# B&R Automation Studio project Inzynierka_Kucharczyk_2018
Automation Studio 4.3.7.46 SP; technology packages: Acp10Arnc0 3.18.2, mapp 1.62.1

## Configuration Config1

CPU 4PP065.0571-P74F, AutomationRuntime G4.34, Build 4.1.2

### Task classes (Cpu.sw)
```
Cyclic#4:
  AxisCtrl <- Source.Code.AxisControl.AxisCtrl.prg
  Program <- Source.Code.Package1.Program.prg
NcDataObjects: acp10etxen <- acp10etxen.dob, gAxis01a <- gAxis01obj.gAxis01a.dob, gAxis01i <- gAxis01obj.gAxis01i.dob
VcDataObjects: Visu <- Source.Visu.Visu.dob
Libraries: MpAxis, MpCom, MpBase, NcGlobal, Acp10_MC, brsystem, Acp10man, sys_lib, Acp10par, runtime
```

### Hardware
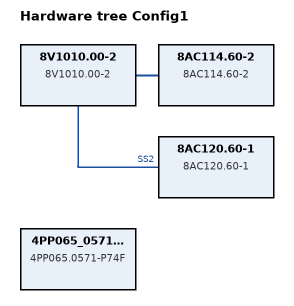
```
4PP065_0571_P74F : 4PP065.0571-P74F v1.0.3.0
  Connector IF5:
    ActivateDevice = 1
  ConfigurationID = Inzynierka_Kucharczyk_2018_Config1
  SimulationInaPort = 5900
  TimerDeviceType = EPLX2X
  TimerDevice = 4PP065_0571_P74F.IF4
  TaskClassIdleTime = 2000
  ActivateOpcUa = 1
  OpcUa_Security_AdminRole = Everyone
  OpcUaInformationModels_PV_Version = 1
  VcObjectName = Visu
  KeyMappingFile = VC\4PP065_0571_P74F.dis
8AC114.60-2 : 8AC114.60-2 v1.0.0.8  [SS -> 8V1010.00-2.SS1; PLK1 -> 4PP065_0571_P74F.IF4 [Cable Type=PowerlinkCable, Length=10, Version=1.0.0.1]]
8AC120.60-1 : 8AC120.60-1 v1.0.0.2  [SS -> 8V1010.00-2.SS2]
8V1010.00-2 : 8V1010.00-2 v1.0.0.2
  PoweredBy = DC
  BothEndSwitchesAreNormallyOpen_r1 = on
  QuickStopIsNormallyOpen_r1 = on
```

### Acp10cfg.ncc - 4PP065_0571_P74F/Motion/Acp10cfg.ncc
```
NcConfiguration (Version=3.18.2, NcSwId=Acp10)
  ACP10CF1_typ:
    cnt_nettrc_rec_drive = 150
    bufsize_trace_upload = 1200
    tc_nc_man_task = Cyclic #1
    glob_pv_as_ncobject = Yes
    ncsys_dl_broadcast = Yes
    ncsys_dl_acp_reset = Yes
    safemc_log_err_to_ax = Yes
    network_init:
      ncsw_init_execute = Yes
      automatic_execute = No
      node_nr_warning = Yes
      net_err_before_ncact = Yes
    nettrc:
      enter_parsecrec = Yes
      enter_ncaction = Yes
      save_ring_startidx = No
    cam_prof_download:
      cam_dat_dl_parallel = No
      tc_cam_dl_parallel = Task class for NC Manager task
    plk_if[0]:
      if_name = IF4
      tc_CycDat_PLCopen = Task class for NC Manager task
      mc_broadcast_extdat = No
```

### Acp10map.ncm - 4PP065_0571_P74F/Motion/Acp10map.ncm
```
NcMapping (NcSwId=Acp10)
  NcObject gAxis01 (ModuleId=8V1010.00-2, Type=ncAXIS, Channel=1, AcoposSimulation=Off, InitParameter=gAxis01i, AcoposParameter=gAxis01a, Disabled=FALSE, ModuleDisabled=FALSE)
  NcObject 8V1010.00-2_ncV_AXIS1 (ModuleId=8V1010.00-2, Type=ncV_AXIS, Channel=1, Disabled=TRUE, ModuleDisabled=FALSE)
```

### Config.mpaxisbasic - 4PP065_0571_P74F/mapp/Config.mpaxisbasic
```
Element gAxisBasic (Type=mpaxisbasic)
  AxisConfiguration = AxisWithConfiguration
    Axis:
      BaseType = 4
      MeasurementUnit = 1
    Drive:
      Controller:
        LoopFilters:
          [0]
          [1]
          [2]
```

## Logical view

Binary libraries used (declarations not repeated): operator, runtime, astime, AsIecCon, MpAxis 1.62.1, MpCom 1.62.1, MpBase 5.00.0, NcGlobal, Acp10_MC, brsystem, Acp10man, sys_lib, Acp10par, Acp10sim 3.18.2, ArEventLog, asstring, FileIO, ArProject

### Global.typ - Global data types
```iecst
TYPE
	Data_OPC_struct : 	STRUCT
		Zmienna1 : USINT;
		Zmienna2 : BOOL;
	END_STRUCT;
END_TYPE
```

### Global.var - Global variables
```iecst
VAR
	Zm_wyj : Data_OPC_struct;
	gAxis01 : ACP10AXIS_typ;
END_VAR
```


### Program Logical/Source/Code/AxisControl/AxisCtrl (IEC)

#### Main.st - Init, cyclic, exit code
```iecst
PROGRAM _INIT
	(* Task to initilization of drives *)
	Initialization;

END_PROGRAM

PROGRAM _CYCLIC

	AxesControl;

	Output_commands;
END_PROGRAM

PROGRAM _EXIT
	ExitAction;

END_PROGRAM
```

#### Initalization.st
```iecst
ACTION Initialization:

	_AxisCtrl.Internal.FunctionsBlock.MpAxisBasic_0.Enable := TRUE;
	_AxisCtrl.Internal.FunctionsBlock.MpAxisBasic_0.Axis   := ADR(gAxis01);
	_AxisCtrl.Internal.FunctionsBlock.MpAxisBasic_0.MpLink := ADR(gAxisBasic);
	_AxisCtrl.Internal.FunctionsBlock.MpAxisBasic_0.Parameters  := ADR(_AxisCtrl.Internal.Functions.MpAxisBasicParType_0);

END_ACTION
```

#### InputCmds.st
```iecst
ACTION Input_commands:

	(* ALL AXIS *)
	IF _AxisCtrl.Input.Commands.AllAxis.PowerOn THEN
		_AxisCtrl.Input.Commands.AllAxis.PowerOn := FALSE;
		_AxisCtrl.Output.Status.AxisStateMachine := POWER_ON;

	ELSIF _AxisCtrl.Input.Commands.AllAxis.PowerOff THEN
		_AxisCtrl.Input.Commands.AllAxis.PowerOff := FALSE;
		_AxisCtrl.Output.Status.AxisStateMachine := POWER_OFF;

	ELSIF _AxisCtrl.Input.Commands.AllAxis.Home THEN
		_AxisCtrl.Input.Commands.AllAxis.Home := FALSE;
		_AxisCtrl.Output.Status.AxisStateMachine := HOME;

	ELSIF _AxisCtrl.Input.Commands.AllAxis.StopOn THEN
		_AxisCtrl.Input.Commands.AllAxis.StopOn := FALSE;
		_AxisCtrl.Output.Status.AxisStateMachine := STOP_ON;

	ELSIF _AxisCtrl.Input.Commands.AllAxis.StopOff THEN
		_AxisCtrl.Input.Commands.AllAxis.StopOff := FALSE;
		_AxisCtrl.Output.Status.AxisStateMachine := STOP_OFF;

	ELSIF _AxisCtrl.Input.Commands.AllAxis.MoveAbsolute THEN
		_AxisCtrl.Input.Commands.AllAxis.MoveAbsolute := FALSE;
		_AxisCtrl.Output.Status.AxisStateMachine := MOVE_ABSOLUTE;

	ELSIF _AxisCtrl.Input.Commands.AllAxis.MoveVelocity THEN
		_AxisCtrl.Input.Commands.AllAxis.MoveVelocity := FALSE;
		_AxisCtrl.Output.Status.AxisStateMachine := MOVE_VELOCITY;

	ELSIF _AxisCtrl.Input.Commands.AllAxis.MoveAdditive THEN
		_AxisCtrl.Input.Commands.AllAxis.MoveAdditive := FALSE;
		_AxisCtrl.Output.Status.AxisStateMachine := MOVE_ADDITIVE;

	ELSIF _AxisCtrl.Input.Commands.AllAxis.JogPositive THEN
		_AxisCtrl.Output.Status.AxisStateMachine := JOG;

	ELSIF _AxisCtrl.Input.Commands.AllAxis.JogNegative THEN
		_AxisCtrl.Output.Status.AxisStateMachine := JOG;

	ELSIF _AxisCtrl.Input.Commands.AllAxis.ErrorReset THEN
		_AxisCtrl.Input.Commands.AllAxis.ErrorReset := FALSE;
		_AxisCtrl.Output.Status.AxisStateMachine := ERROR_RESET;

	(* SINGLE AXIS *)
	ELSIF _AxisCtrl.Input.Commands.SingleAxis.PowerOn THEN
		_AxisCtrl.Input.Commands.SingleAxis.PowerOn := FALSE;
		_AxisCtrl.Output.Status.AxisStateMachine := POWER_ON;

	ELSIF _AxisCtrl.Input.Commands.SingleAxis.PowerOff THEN
		_AxisCtrl.Input.Commands.SingleAxis.PowerOff := FALSE;
		_AxisCtrl.Output.Status.AxisStateMachine := POWER_OFF;

	ELSIF _AxisCtrl.Input.Commands.SingleAxis.Home THEN
		_AxisCtrl.Input.Commands.SingleAxis.Home := FALSE;
		_AxisCtrl.Output.Status.AxisStateMachine := HOME;

	ELSIF _AxisCtrl.Input.Commands.SingleAxis.StopOn THEN
		_AxisCtrl.Input.Commands.SingleAxis.StopOn := FALSE;
		_AxisCtrl.Output.Status.AxisStateMachine := STOP_ON;

	ELSIF _AxisCtrl.Input.Commands.SingleAxis.StopOff THEN
		_AxisCtrl.Input.Commands.SingleAxis.StopOff := FALSE;
		_AxisCtrl.Output.Status.AxisStateMachine := STOP_OFF;

	ELSIF _AxisCtrl.Input.Commands.SingleAxis.MoveAbsolute THEN
		_AxisCtrl.Input.Commands.SingleAxis.MoveAbsolute := FALSE;
		_AxisCtrl.Output.Status.AxisStateMachine := MOVE_ABSOLUTE;

	ELSIF _AxisCtrl.Input.Commands.SingleAxis.MoveVelocity THEN
		_AxisCtrl.Input.Commands.SingleAxis.MoveVelocity := FALSE;
		_AxisCtrl.Output.Status.AxisStateMachine := MOVE_VELOCITY;

	ELSIF _AxisCtrl.Input.Commands.SingleAxis.MoveAdditive THEN
		_AxisCtrl.Input.Commands.SingleAxis.MoveAdditive := FALSE;
		_AxisCtrl.Output.Status.AxisStateMachine := MOVE_ADDITIVE;

	ELSIF _AxisCtrl.Input.Commands.SingleAxis.JogPositive THEN
		_AxisCtrl.Output.Status.AxisStateMachine := JOG;

	ELSIF _AxisCtrl.Input.Commands.SingleAxis.JogNegative THEN
		_AxisCtrl.Output.Status.AxisStateMachine := JOG;

	ELSIF _AxisCtrl.Input.Commands.SingleAxis.ErrorReset THEN
		_AxisCtrl.Input.Commands.SingleAxis.ErrorReset := FALSE;
		_AxisCtrl.Output.Status.AxisStateMachine := ERROR_RESET;

	END_IF

END_ACTION
```

#### AxisControl.st
```iecst
ACTION AxesControl:

	CASE _AxisCtrl.Output.Status.AxisStateMachine OF
		WAIT_FOR_CMD:

			Input_commands;

		WAIT_FOR_ACTIVE:

		POWER_ON:

		POWER_OFF:

		HOME:

		STOP_ON:

		STOP_OFF:

		MOVE_ABSOLUTE:

		MOVE_VELOCITY:

		MOVE_ADDITIVE:

		JOG:

		ERROR_RESET:

	END_CASE;

END_ACTION
```

#### OutputCmds.st
```iecst
ACTION Output_commands:
	(* ALL AXES *)
	_AxisCtrl.Output.States.AllAxis.Active  := _AxisCtrl.Internal.FunctionsBlock.MpAxisBasic_0.Active;
	_AxisCtrl.Output.States.AllAxis.PowerOn := _AxisCtrl.Internal.FunctionsBlock.MpAxisBasic_0.PowerOn;
	_AxisCtrl.Output.States.AllAxis.IsHomed := _AxisCtrl.Internal.FunctionsBlock.MpAxisBasic_0.IsHomed;
	_AxisCtrl.Output.States.AllAxis.Stopped := _AxisCtrl.Internal.FunctionsBlock.MpAxisBasic_0.Stopped;
	_AxisCtrl.Output.States.AllAxis.InPosition := _AxisCtrl.Internal.FunctionsBlock.MpAxisBasic_0.InPosition;
	_AxisCtrl.Output.States.AllAxis.InVelocity := _AxisCtrl.Internal.FunctionsBlock.MpAxisBasic_0.InVelocity;
	_AxisCtrl.Output.States.AllAxis.MoveActive := _AxisCtrl.Internal.FunctionsBlock.MpAxisBasic_0.MoveActive;
	_AxisCtrl.Output.States.AllAxis.Error 	   := _AxisCtrl.Internal.FunctionsBlock.MpAxisBasic_0.Error;

	(* FIRST AXIS *)
	_AxisCtrl.Output.States.SingleAxis.Axis_0.Active  := _AxisCtrl.Internal.FunctionsBlock.MpAxisBasic_0.Active;
	_AxisCtrl.Output.States.SingleAxis.Axis_0.PowerOn := _AxisCtrl.Internal.FunctionsBlock.MpAxisBasic_0.PowerOn;
	_AxisCtrl.Output.States.SingleAxis.Axis_0.IsHomed := _AxisCtrl.Internal.FunctionsBlock.MpAxisBasic_0.IsHomed;
	_AxisCtrl.Output.States.SingleAxis.Axis_0.Stopped := _AxisCtrl.Internal.FunctionsBlock.MpAxisBasic_0.Stopped;
	_AxisCtrl.Output.States.SingleAxis.Axis_0.InPosition := _AxisCtrl.Internal.FunctionsBlock.MpAxisBasic_0.InPosition;
	_AxisCtrl.Output.States.SingleAxis.Axis_0.InVelocity := _AxisCtrl.Internal.FunctionsBlock.MpAxisBasic_0.InVelocity;
	_AxisCtrl.Output.States.SingleAxis.Axis_0.MoveActive := _AxisCtrl.Internal.FunctionsBlock.MpAxisBasic_0.MoveActive;
	_AxisCtrl.Output.States.SingleAxis.Axis_0.Error		 := _AxisCtrl.Internal.FunctionsBlock.MpAxisBasic_0.Error;
	_AxisCtrl.Output.States.SingleAxis.Axis_0.StatusID	 := _AxisCtrl.Internal.FunctionsBlock.MpAxisBasic_0.StatusID;

_AxisCtrl.Internal.FunctionsBlock.MpAxisBasic_0();
END_ACTION
```

#### Exit.st
```iecst
ACTION ExitAction:

END_ACTION
```

#### Axis1.st - not listed in the package file held
```iecst
ACTION Axis1:

	CASE _AxisCtrl.Output.Status.AxisStateMachine OF
		WAIT_FOR_CMD:

			IF _AxisCtrl.Input.Commands.SingleAxis.A1.PowerOn THEN
				_AxisCtrl.Input.Commands.SingleAxis.A1.PowerOn := FALSE;
				_AxisCtrl.Output.Status.AxisStateMachine := POWER_ON;

			ELSIF _AxisCtrl.Input.Commands.SingleAxis.A1.PowerOff THEN
				_AxisCtrl.Input.Commands.SingleAxis.A1.PowerOff := FALSE;
				_AxisCtrl.Output.Status.AxisStateMachine := POWER_OFF;

			ELSIF _AxisCtrl.Input.Commands.SingleAxis.A1.Home THEN
				_AxisCtrl.Input.Commands.SingleAxis.A1.Home := FALSE;
				_AxisCtrl.Output.Status.HomingStateMachine := PREPARE_HOME;
				_AxisCtrl.Output.Status.AxisStateMachine := HOME;

			ELSIF _AxisCtrl.Input.Commands.SingleAxis.A1.StopOn THEN
				_AxisCtrl.Input.Commands.SingleAxis.A1.StopOn := FALSE;
				_AxisCtrl.Output.Status.AxisStateMachine := STOP_ON;

			ELSIF _AxisCtrl.Input.Commands.SingleAxis.A1.StopOff THEN
				_AxisCtrl.Input.Commands.SingleAxis.A1.StopOff := FALSE;
				_AxisCtrl.Output.Status.AxisStateMachine := STOP_OFF;

			ELSIF _AxisCtrl.Input.Commands.SingleAxis.A1.MoveAbsolute THEN
				_AxisCtrl.Input.Commands.SingleAxis.A1.MoveAbsolute := FALSE;
				_AxisCtrl.Output.Status.AxisStateMachine := MOVE_ABSOLUTE;

			ELSIF _AxisCtrl.Input.Commands.SingleAxis.A1.MoveAbsoluteOff THEN
				_AxisCtrl.Input.Commands.SingleAxis.A1.MoveAbsoluteOff := FALSE;
				_AxisCtrl.Output.Status.AxisStateMachine := MOVE_ABSOLUTE_OFF;

			ELSIF _AxisCtrl.Input.Commands.SingleAxis.A1.MoveVelocity THEN
				_AxisCtrl.Input.Commands.SingleAxis.A1.MoveVelocity := FALSE;
				_AxisCtrl.Output.Status.AxisStateMachine := MOVE_VELOCITY;

			ELSIF _AxisCtrl.Input.Commands.SingleAxis.A1.MoveVelocityOff THEN
				_AxisCtrl.Input.Commands.SingleAxis.A1.MoveVelocityOff := FALSE;
				_AxisCtrl.Output.Status.AxisStateMachine := MOVE_VELOCITY_OFF;

			ELSIF _AxisCtrl.Input.Commands.SingleAxis.A1.MoveAdditive THEN
				_AxisCtrl.Input.Commands.SingleAxis.A1.MoveAdditive := FALSE;
				_AxisCtrl.Output.Status.AxisStateMachine := MOVE_ADDITIVE;

			ELSIF _AxisCtrl.Input.Commands.SingleAxis.A1.MoveAdditiveOff THEN
				_AxisCtrl.Input.Commands.SingleAxis.A1.MoveAdditiveOff := FALSE;
				_AxisCtrl.Output.Status.AxisStateMachine := MOVE_ADDITIVE_OFF;

			ELSIF _AxisCtrl.Input.Commands.SingleAxis.A1.JogPositive THEN
				_AxisCtrl.Output.Status.AxisStateMachine := JOG_POSITIVE;

			ELSIF _AxisCtrl.Input.Commands.SingleAxis.A1.JogNegative THEN
				_AxisCtrl.Output.Status.AxisStateMachine := JOG_NEGATIVE;

			ELSIF _AxisCtrl.Input.Commands.SingleAxis.A1.Update THEN
				_AxisCtrl.Input.Commands.SingleAxis.A1.Update := FALSE;
				_AxisCtrl.Internal.Functions.MpAxisBasicParType_0.Acceleration := _AxisCtrl.Input.Parameters.Acceleration;
				_AxisCtrl.Internal.Functions.MpAxisBasicParType_0.Deceleration := _AxisCtrl.Input.Parameters.Deceleration;
				_AxisCtrl.Internal.Functions.MpAxisBasicParType_0.Distance	   := _AxisCtrl.Input.Parameters.Distance;
				_AxisCtrl.Internal.Functions.MpAxisBasicParType_0.Position 	   := _AxisCtrl.Input.Parameters.Position;
				_AxisCtrl.Internal.Functions.MpAxisBasicParType_0.Velocity 	   := _AxisCtrl.Input.Parameters.Velocity;
			//	_AxisCtrl.Internal.Functions.MpAxisBasicParType_0.Torque.Limit  := _AxisCtrl.Input.Parameters.TorqueLimit;
			//	_AxisCtrl.Internal.Functions.MpAxisBasicParType_0.Torque.Window := _AxisCtrl.Input.Parameters.TorqueWindow;

				_AxisCtrl.Output.Status.AxisStateMachine := UPDATE_MP_AXIS_BASIC;

			ELSIF _AxisCtrl.Input.Commands.SingleAxis.A1.UpdateJogParams THEN
				_AxisCtrl.Input.Commands.SingleAxis.A1.UpdateJogParams := FALSE;
				_AxisCtrl.Internal.Functions.MpAxisBasicParType_0.Jog.Acceleration := _AxisCtrl.Input.Parameters.JogParams.Acceleration;
				_AxisCtrl.Internal.Functions.MpAxisBasicParType_0.Jog.Deceleration := _AxisCtrl.Input.Parameters.JogParams.Deceleration;
				_AxisCtrl.Internal.Functions.MpAxisBasicParType_0.Jog.LowerLimit   := _AxisCtrl.Input.Parameters.JogParams.LowerLimit;
			//	_AxisCtrl.Internal.Functions.MpAxisBasicParType_0.Jog.UpperLimit   := _AxisCtrl.Input.Parameters.JogParams.UpperLimit;
				_AxisCtrl.Internal.Functions.MpAxisBasicParType_0.Jog.Velocity     := _AxisCtrl.Input.Parameters.JogParams.JogVelocity;

				_AxisCtrl.Output.Status.AxisStateMachine := UPDATE_JOG_PARAMS;

				(* CYCLIC SET FUBS *)
			ELSIF _AxisCtrl.Input.Commands.SingleAxis.A1.TorqControl.CyclicPositionOn THEN
				_AxisCtrl.Input.Commands.SingleAxis.A1.TorqControl.CyclicPositionOn := FALSE;
				_AxisCtrl.Output.Status.AxisStateMachine := CYCLIC_POSITION_ON;

			ELSIF _AxisCtrl.Input.Commands.SingleAxis.A1.TorqControl.CyclicTorqueOn THEN
				_AxisCtrl.Input.Commands.SingleAxis.A1.TorqControl.CyclicTorqueOff := FALSE;
				_AxisCtrl.Output.Status.AxisStateMachine := CYCLIC_TORQUE_ON;

			ELSIF _AxisCtrl.Input.Commands.SingleAxis.A1.TorqControl.CyclicVelocityOn THEN
				_AxisCtrl.Input.Commands.SingleAxis.A1.TorqControl.CyclicVelocityOff := FALSE;
				_AxisCtrl.Output.Status.AxisStateMachine := CYCLIC_VELOCITY_ON;

			ELSIF _AxisCtrl.Input.Commands.SingleAxis.A1.TorqControl.CyclicPositionOff THEN
				_AxisCtrl.Input.Commands.SingleAxis.A1.TorqControl.CyclicPositionOff := FALSE;
				_AxisCtrl.Output.Status.AxisStateMachine := CYCLIC_POSITION_OFF;

			ELSIF _AxisCtrl.Input.Commands.SingleAxis.A1.TorqControl.CyclicTorqueOff THEN
				_AxisCtrl.Input.Commands.SingleAxis.A1.TorqControl.CyclicTorqueOff := FALSE;
				_AxisCtrl.Output.Status.AxisStateMachine := CYCLIC_TORQUE_OFF;

			ELSIF _AxisCtrl.Input.Commands.SingleAxis.A1.TorqControl.CyclicVelocityOff THEN
				_AxisCtrl.Input.Commands.SingleAxis.A1.TorqControl.CyclicVelocityOff := FALSE;
				_AxisCtrl.Output.Status.AxisStateMachine := CYCLIC_VELOCITY_OFF;

			ELSIF _AxisCtrl.Input.Commands.SingleAxis.A1.TorqControl.Update THEN

				_AxisCtrl.Internal.FunctionsBlock.TorqueControl.Position := _AxisCtrl.Input.Parameters.CyclicSetParameter.Position;
				_AxisCtrl.Internal.FunctionsBlock.TorqueControl.Torque 	 := _AxisCtrl.Input.Parameters.CyclicSetParameter.Torque;
				_AxisCtrl.Internal.FunctionsBlock.TorqueControl.Velocity := _AxisCtrl.Input.Parameters.CyclicSetParameter.Velocity;

				_AxisCtrl.Input.Commands.SingleAxis.A1.TorqControl.Update := FALSE;
				_AxisCtrl.Output.Status.AxisStateMachine := UPDATE_CYCLIC_SET;

			END_IF

		WAIT_FOR_ACTIVE:
			IF _AxisCtrl.Internal.FunctionsBlock.MpAxisBasic_0.Active THEN
				_AxisCtrl.Output.Status.AxisStateMachine := WAIT_FOR_CMD;
			ELSIF _AxisCtrl.Internal.FunctionsBlock.MpAxisBasic_0.Error THEN
				_AxisCtrl.Output.Status.AxisStateMachine := ERROR;
			END_IF

		POWER_ON:
			IF _AxisCtrl.Internal.FunctionsBlock.MpAxisBasic_0.PowerOn THEN
				_AxisCtrl.Output.Status.AxisStateMachine := WAIT_FOR_CMD;

			ELSIF _AxisCtrl.Internal.FunctionsBlock.MpAxisBasic_0.Error THEN
				_AxisCtrl.Internal.FunctionsBlock.MpAxisBasic_0.Power := FALSE;
				_AxisCtrl.Output.Status.AxisStateMachine := ERROR;

			ELSE
				_AxisCtrl.Internal.FunctionsBlock.MpAxisBasic_0.Power := TRUE;

			END_IF

		POWER_OFF:
			IF NOT _AxisCtrl.Internal.FunctionsBlock.MpAxisBasic_0.PowerOn THEN
				_AxisCtrl.Output.Status.AxisStateMachine := WAIT_FOR_CMD;

			ELSIF _AxisCtrl.Internal.FunctionsBlock.MpAxisBasic_0.Error THEN
				_AxisCtrl.Internal.FunctionsBlock.MpAxisBasic_0.Power := FALSE;
				_AxisCtrl.Output.Status.AxisStateMachine := ERROR;

			ELSE
				_AxisCtrl.Internal.FunctionsBlock.MpAxisBasic_0.Power := FALSE;
			END_IF

		HOME:
			CASE _AxisCtrl.Output.Status.HomingStateMachine OF
				PREPARE_HOME:
					_AxisCtrl.Internal.FunctionsBlock.MpAxisBasic_0.Home := FALSE;
					_AxisCtrl.Output.Status.HomingStateMachine := HOMING;
				HOMING:
					_AxisCtrl.Internal.FunctionsBlock.MpAxisBasic_0.Home := TRUE;
					IF _AxisCtrl.Internal.FunctionsBlock.MpAxisBasic_0.IsHomed THEN
						_AxisCtrl.Internal.FunctionsBlock.MpAxisBasic_0.Home := FALSE;
						_AxisCtrl.Output.Status.HomingStateMachine := EXIT_HOME;
					END_IF
				EXIT_HOME:
					_AxisCtrl.Output.Status.AxisStateMachine := WAIT_FOR_CMD;
					_AxisCtrl.Output.Status.HomingStateMachine := PREPARE_HOME;
			END_CASE;

		STOP_ON:
			IF _AxisCtrl.Internal.FunctionsBlock.MpAxisBasic_0.Stopped THEN
				_AxisCtrl.Output.Status.AxisStateMachine := WAIT_FOR_CMD;
			ELSIF _AxisCtrl.Internal.FunctionsBlock.MpAxisBasic_0.Error THEN
				_AxisCtrl.Internal.FunctionsBlock.MpAxisBasic_0.Stop := FALSE;
				_AxisCtrl.Output.Status.AxisStateMachine := ERROR;
			ELSE
				_AxisCtrl.Internal.FunctionsBlock.MpAxisBasic_0.Stop := TRUE;
			END_IF

		STOP_OFF:
			IF NOT _AxisCtrl.Internal.FunctionsBlock.MpAxisBasic_0.Stopped THEN
				_AxisCtrl.Output.Status.AxisStateMachine := WAIT_FOR_CMD;
			ELSIF _AxisCtrl.Internal.FunctionsBlock.MpAxisBasic_0.Error THEN
				_AxisCtrl.Internal.FunctionsBlock.MpAxisBasic_0.Stop := FALSE;
				_AxisCtrl.Output.Status.AxisStateMachine := ERROR;
			ELSE
				_AxisCtrl.Internal.FunctionsBlock.MpAxisBasic_0.Stop := FALSE;
			END_IF

		MOVE_ABSOLUTE:

			_AxisCtrl.Internal.FunctionsBlock.MpAxisBasic_0.MoveAbsolute := TRUE;
			_AxisCtrl.Output.Status.AxisStateMachine := WAIT_FOR_CMD;

		MOVE_ABSOLUTE_OFF:

			_AxisCtrl.Internal.FunctionsBlock.MpAxisBasic_0.MoveAbsolute := FALSE;
			_AxisCtrl.Output.Status.AxisStateMachine := WAIT_FOR_CMD;

		MOVE_VELOCITY:

			_AxisCtrl.Internal.FunctionsBlock.MpAxisBasic_0.MoveVelocity := TRUE;
			_AxisCtrl.Output.Status.AxisStateMachine := WAIT_FOR_CMD;

		MOVE_VELOCITY_OFF:

			_AxisCtrl.Internal.FunctionsBlock.MpAxisBasic_0.MoveVelocity := FALSE;
			_AxisCtrl.Output.Status.AxisStateMachine := WAIT_FOR_CMD;

		MOVE_ADDITIVE:

			_AxisCtrl.Internal.FunctionsBlock.MpAxisBasic_0.MoveAdditive := TRUE;
			_AxisCtrl.Output.Status.AxisStateMachine := WAIT_FOR_CMD;

		MOVE_ADDITIVE_OFF:

			_AxisCtrl.Internal.FunctionsBlock.MpAxisBasic_0.MoveAdditive := FALSE;
			_AxisCtrl.Output.Status.AxisStateMachine := WAIT_FOR_CMD;

		JOG_POSITIVE:
			IF NOT _AxisCtrl.Input.Commands.SingleAxis.A1.JogPositive THEN
				_AxisCtrl.Internal.FunctionsBlock.MpAxisBasic_0.JogPositive := FALSE;
				_AxisCtrl.Output.Status.AxisStateMachine := WAIT_FOR_CMD;
			ELSE
				_AxisCtrl.Internal.FunctionsBlock.MpAxisBasic_0.JogPositive := TRUE;
			END_IF

		JOG_NEGATIVE:
			IF NOT _AxisCtrl.Input.Commands.SingleAxis.A1.JogNegative THEN
				_AxisCtrl.Internal.FunctionsBlock.MpAxisBasic_0.JogNegative := FALSE;
				_AxisCtrl.Output.Status.AxisStateMachine := WAIT_FOR_CMD;
			ELSE
				_AxisCtrl.Internal.FunctionsBlock.MpAxisBasic_0.JogNegative := TRUE;
			END_IF

		UPDATE_MP_AXIS_BASIC:
			IF _AxisCtrl.Internal.FunctionsBlock.MpAxisBasic_0.UpdateDone THEN
				_AxisCtrl.Internal.FunctionsBlock.MpAxisBasic_0.Update := FALSE;
				_AxisCtrl.Output.Status.AxisStateMachine := WAIT_FOR_CMD;
			ELSE
				_AxisCtrl.Internal.FunctionsBlock.MpAxisBasic_0.Update := TRUE;
			END_IF

		UPDATE_JOG_PARAMS:
			IF _AxisCtrl.Internal.FunctionsBlock.MpAxisBasic_0.UpdateDone THEN
				_AxisCtrl.Internal.FunctionsBlock.MpAxisBasic_0.Update := FALSE;
				_AxisCtrl.Output.Status.AxisStateMachine := WAIT_FOR_CMD;
			ELSE
				_AxisCtrl.Internal.FunctionsBlock.MpAxisBasic_0.Update := TRUE;
			END_IF

		ERROR:
			IF _AxisCtrl.Input.Commands.SingleAxis.A1.ErrorReset OR _AxisCtrl.Input.Commands.SingleAxis.A1.TorqControl.ErrorReset THEN
				_AxisCtrl.Internal.FunctionsBlock.MpAxisBasic_0.ErrorReset := TRUE;
				_AxisCtrl.Internal.FunctionsBlock.TorqueControl.ErrorReset := TRUE;
				_AxisCtrl.Output.Status.AxisStateMachine := ERROR_RESET;
			END_IF

		ERROR_RESET:
			IF NOT _AxisCtrl.Output.States.SingleAxis.Axis_0.Error AND NOT _AxisCtrl.Internal.FunctionsBlock.TorqueControl.Error THEN
				_AxisCtrl.Internal.FunctionsBlock.MpAxisBasic_0.ErrorReset := FALSE;
				_AxisCtrl.Internal.FunctionsBlock.TorqueControl.ErrorReset := FALSE;
				_AxisCtrl.Output.Status.AxisStateMachine := WAIT_FOR_CMD;

			END_IF

		CYCLIC_POSITION_ON:

	    		_AxisCtrl.Internal.FunctionsBlock.TorqueControl.CyclicPosition := TRUE;
				_AxisCtrl.Output.Status.AxisStateMachine := WAIT_FOR_CMD;

		CYCLIC_POSITION_OFF:

				_AxisCtrl.Internal.FunctionsBlock.TorqueControl.CyclicPosition := FALSE;
				_AxisCtrl.Output.Status.AxisStateMachine := WAIT_FOR_CMD;

		CYCLIC_TORQUE_ON:

			_AxisCtrl.Internal.FunctionsBlock.TorqueControl.CyclicTorque := TRUE;
			_AxisCtrl.Output.Status.AxisStateMachine := WAIT_FOR_CMD;

		CYCLIC_TORQUE_OFF:

			_AxisCtrl.Internal.FunctionsBlock.TorqueControl.CyclicTorque := FALSE;
			_AxisCtrl.Output.Status.AxisStateMachine := WAIT_FOR_CMD;

		CYCLIC_VELOCITY_ON:

			_AxisCtrl.Internal.FunctionsBlock.TorqueControl.CyclicVelocity := TRUE;
			_AxisCtrl.Output.Status.AxisStateMachine := WAIT_FOR_CMD;

		CYCLIC_VELOCITY_OFF:

			_AxisCtrl.Internal.FunctionsBlock.TorqueControl.CyclicVelocity := FALSE;
			_AxisCtrl.Output.Status.AxisStateMachine := WAIT_FOR_CMD;

		UPDATE_CYCLIC_SET:
			IF _AxisCtrl.Internal.FunctionsBlock.TorqueControl.UpdateDone THEN
				_AxisCtrl.Internal.FunctionsBlock.TorqueControl.Update := FALSE;
				_AxisCtrl.Output.Status.AxisStateMachine := WAIT_FOR_CMD;
			ELSE
				_AxisCtrl.Internal.FunctionsBlock.TorqueControl.Update := TRUE;
			END_IF

	END_CASE;

END_ACTION
```

#### Axis2.st - not listed in the package file held
```iecst
ACTION Axis2:

END_ACTION
```

#### ErrorHandling.st - not listed in the package file held
```iecst
ACTION ErrorHandling:

	IF (_AxisCtrl.Internal.FunctionsBlock.MpAxisBasic_0.Error OR _AxisCtrl.Internal.FunctionsBlock.TorqueControl.Error) AND _AxisCtrl.Output.Status.AxisStateMachine <> ERROR_RESET THEN
		_AxisCtrl.Output.Status.AxisStateMachine := ERROR;
	END_IF

END_ACTION
```

#### Types.typ - Local data types
```iecst
(*Main structure*)

TYPE
	AxisCtrlType : 	STRUCT
		Input : AxisCtrlInpType; (*Inputs: ex. commands*)
		Internal : AxisCtrlInternalType; (*Fubs, funs*)
		Output : AxisCtrlOutType; (*States, status*)
	END_STRUCT;
END_TYPE

(**)
(*Inputs*)

TYPE
	AxisCtrlInpType : 	STRUCT
		Commands : {REDUND_UNREPLICABLE} AxisCtrlInpCmdType;
		Parameters : AxisCtrlInpParamsType;
	END_STRUCT;
END_TYPE

(**)

TYPE
	AxisCtrlInpCmdType : 	STRUCT
		SingleAxis : AxisCtrlInpCmdSigAxType;
		AllAxis : AxisCtrlInpCmdAllAxType;
	END_STRUCT;
	AxisCtrlInpParamsType : 	STRUCT
		Acceleration : REAL;
		Deceleration : REAL;
		Distance : REAL;
		Velocity : REAL;
		Position : REAL;
		JogParams : AxisCtrlInpParmsJogPType;
	END_STRUCT;
END_TYPE

(**)

TYPE
	AxisCtrlInpCmdSigAxType : 	STRUCT
		PowerOn : BOOL;
		PowerOff : BOOL;
		Home : BOOL;
		MoveVelocity : BOOL;
		MoveAdditive : BOOL;
		MoveAbsolute : BOOL;
		StopOn : BOOL;
		StopOff : BOOL;
		JogNegative : BOOL;
		JogPositive : BOOL;
		ErrorReset : BOOL;
	END_STRUCT;
	AxisCtrlInpCmdAllAxType : 	STRUCT
		PowerOn : BOOL;
		PowerOff : BOOL;
		Home : BOOL;
		MoveVelocity : BOOL;
		MoveAdditive : BOOL;
		MoveAbsolute : BOOL;
		StopOn : BOOL;
		StopOff : BOOL;
		JogNegative : BOOL;
		JogPositive : BOOL;
		ErrorReset : BOOL;
	END_STRUCT;
	AxisCtrlInpParmsJogPType : 	STRUCT
		JogVelocity : REAL;
		Acceleration : REAL;
		Deceleration : REAL;
		UpperLimit : LREAL;
		LowerLimit : LREAL;
	END_STRUCT;
END_TYPE

(**)
(*Internal*)

TYPE
	AxisCtrlInternalType : 	STRUCT
		FunctionsBlock : AxisCtrlInternalFubsType;
		Functions : AxisCtrlInternalFunsType;
	END_STRUCT;
END_TYPE

(**)

TYPE
	AxisCtrlInternalFubsType : 	STRUCT
		MpAxisBasic_0 : MpAxisBasic;
	END_STRUCT;
	AxisCtrlInternalFunsType : 	STRUCT
		MpAxisBasicParType_0 : MpAxisBasicParType;
	END_STRUCT;
END_TYPE

(**)
(*Output*)

TYPE
	AxisCtrlOutType : 	STRUCT
		Status : AxisCtrlOutStatusType;
		States : AxisCtrlOutStatesType;
	END_STRUCT;
	AxisCtrlOutStatusType : 	STRUCT
		HomingStateMachine : HomingEnum;
		AxisStateMachine : AxisCtrlEnum;
	END_STRUCT;
	AxisCtrlOutStatesType : 	STRUCT
		SingleAxis : AxisCtrlOutStatesSingType;
		AllAxis : AxisCtrlOutStatesAllType;
	END_STRUCT;
END_TYPE

(**)

TYPE
	AxisCtrlOutStatesAllType : 	STRUCT
		InPosition : BOOL;
		InVelocity : BOOL;
		UpdateDone : BOOL;
		Active : BOOL;
		Error : BOOL;
		Stopped : BOOL;
		MoveActive : BOOL;
		IsHomed : BOOL;
		PowerOn : BOOL;
	END_STRUCT;
	AxisCtrlOutStatesSingType : 	STRUCT
		Axis_0 : AxisCtrlOutStatesSingAxType;
		Axis_1 : AxisCtrlOutStatesSingAxType;
	END_STRUCT;
	AxisCtrlOutStatesSingAxType : 	STRUCT
		InPosition : BOOL;
		InVelocity : BOOL;
		StatusID : DINT;
		UpdateDone : BOOL;
		Active : BOOL;
		Error : BOOL;
		Stopped : BOOL;
		MoveActive : BOOL;
		IsHomed : BOOL;
		PowerOn : BOOL;
	END_STRUCT;
END_TYPE

(**)
(*Enumerators*)

TYPE
	HomingEnum :
		(
		PREPARE_HOME,
		HOMING,
		EXIT_HOME
		);
	AxisCtrlEnum :
		(
		WAIT_FOR_CMD,
		JOG,
		MOVE_ADDITIVE,
		MOVE_VELOCITY,
		MOVE_ABSOLUTE,
		STOP_OFF,
		STOP_ON,
		HOME,
		POWER_OFF,
		POWER_ON,
		WAIT_FOR_ACTIVE,
		ERROR_RESET
		);
END_TYPE
```

#### Variables.var - Local variables
```iecst
VAR
	_AxisCtrl : AxisCtrlType;
END_VAR
```

### Types.typ - not listed in the package file held
```iecst
(*Main structure*)

TYPE
	AxisCtrlType : 	STRUCT
		Input : AxisCtrlInpType; (*Inputs: ex. commands*)
		Internal : AxisCtrlInternalType; (*Fubs, funs*)
		Output : AxisCtrlOutType; (*States, status*)
	END_STRUCT;
END_TYPE

(**)
(*Inputs*)

TYPE
	AxisCtrlInpType : 	STRUCT
		Commands : {REDUND_UNREPLICABLE} AxisCtrlInpCmdType;
		Parameters : AxisCtrlInpParamsType;
	END_STRUCT;
END_TYPE

(**)

TYPE
	AxisCtrlInpCmdType : 	STRUCT
		SingleAxis : AxisCtrlInpCmdSigAxType;
		AllAxis : AxisCtrlInpCmdAllAxType;
	END_STRUCT;
	AxisCtrlInpParamsType : 	STRUCT
		Acceleration : REAL;
		Deceleration : REAL;
		Distance : REAL;
		Velocity : REAL;
		TorqueLimit : REAL;
		Position : REAL;
		TorqueWindow : REAL;
		JogParams : AxisCtrlInpParmsJogPType;
	END_STRUCT;
END_TYPE

(**)

TYPE
	AxisCtrlInpCmdSigAxType : 	STRUCT
		A1 : AxisCtrlInpCmdSingAxAType;
	END_STRUCT;
	AxisCtrlInpCmdSingAxAType : 	STRUCT
		PowerOn : BOOL;
		PowerOff : BOOL;
		Home : BOOL;
		MoveVelocity : BOOL;
		MoveAdditive : BOOL;
		MoveOff : BOOL;
		MoveAbsolute : BOOL;
		MoveTorque : BOOL;
		StopOn : BOOL;
		StopOff : BOOL;
		JogPositive : BOOL;
		JogNegative : BOOL;
		ErrorReset : BOOL;
		Update : BOOL;
	END_STRUCT;
	AxisCtrlInpCmdAllAxType : 	STRUCT
		PowerOn : BOOL;
		PowerOff : BOOL;
		Home : BOOL;
		MoveVelocity : BOOL;
		MoveAdditive : BOOL;
		MoveAbsolute : BOOL;
		MoveTorque : BOOL;
		StopOn : BOOL;
		StopOff : BOOL;
		Jog : BOOL;
		ErrorReset : BOOL;
	END_STRUCT;
	AxisCtrlInpParmsJogPType : 	STRUCT
		JogVelocity : REAL;
		Acceleration : REAL;
		Deceleration : REAL;
		UpperLimit : LREAL;
		LowerLimit : LREAL;
	END_STRUCT;
END_TYPE

(**)
(*Internal*)

TYPE
	AxisCtrlInternalType : 	STRUCT
		FunctionsBlock : AxisCtrlInternalFubsType;
		Functions : AxisCtrlInternalFunsType;
	END_STRUCT;
END_TYPE

(**)

TYPE
	AxisCtrlInternalFubsType : 	STRUCT
		TorqueControl : MpAxisCyclicSet;
		MpAxisBasic_0 : MpAxisBasic;
	END_STRUCT;
	AxisCtrlInternalFunsType : 	STRUCT
		MpTorqueParams : MpAxisCyclicSetParType;
		MpAxisBasicParType_0 : MpAxisBasicParType;
	END_STRUCT;
END_TYPE

(**)
(*Output*)

TYPE
	AxisCtrlOutType : 	STRUCT
		Status : AxisCtrlOutStatusType;
		States : AxisCtrlOutStatesType;
	END_STRUCT;
	AxisCtrlOutStatusType : 	STRUCT
		HomingStateMachine : HomingEnum;
		AxisStateMachine : AxisCtrlEnum;
	END_STRUCT;
	AxisCtrlOutStatesType : 	STRUCT
		SingleAxis : AxisCtrlOutStatesSingType;
		AllAxis : AxisCtrlOutStatesAllType;
		Diagnosis : AxisCtrlOutStatesDiagType;
	END_STRUCT;
END_TYPE

(**)

TYPE
	AxisCtrlOutStatesAllType : 	STRUCT
		InPosition : BOOL;
		InVelocity : BOOL;
		UpdateDone : BOOL;
		Active : BOOL;
		Error : BOOL;
		Stopped : BOOL;
		MoveActive : BOOL;
		IsHomed : BOOL;
		PowerOn : BOOL;
	END_STRUCT;
	AxisCtrlOutStatesSingType : 	STRUCT
		Axis_0 : AxisCtrlOutStatesSingAxType;
		Axis_1 : AxisCtrlOutStatesSingAxType;
	END_STRUCT;
	AxisCtrlOutStatesSingAxType : 	STRUCT
		InPosition : BOOL;
		InVelocity : BOOL;
		StatusID : DINT;
		UpdateDone : BOOL;
		Active : BOOL;
		Error : BOOL;
		Stopped : BOOL;
		MoveActive : BOOL;
		IsHomed : BOOL;
		PowerOn : BOOL;
		Params : AxisCtrlOutStatesSingAxParType;
	END_STRUCT;
	AxisCtrlOutStatesSingAxParType : 	STRUCT
		PositionAct : LREAL;
		Deceleration : LREAL;
		Acceleration : LREAL;
		Position : LREAL;
		TorqueLimit : LREAL;
		Distance : LREAL;
		Velocity : LREAL;
		VelocityAct : LREAL;
	END_STRUCT;
	AxisCtrlOutStatesDiagType : 	STRUCT
		A0 : AxisCtrlOutStatesDiagAxType;
	END_STRUCT;
	AxisCtrlOutStatesDiagAxType : 	STRUCT
		DriveRestarted : BOOL;
		TorqueLimitActive : BOOL;
		JogLimited : BOOL;
		AxisInitialized : BOOL;
		ReadyToOPowerOn : BOOL;
		PLCopenStateAx0 : STRING[80];
	END_STRUCT;
END_TYPE

(**)
(*Enumerators*)

TYPE
	AxisCtrlEnum :
		(
		WAIT_FOR_CMD,
		JOG_NEGATIVE,
		JOG_POSITIVE,
		MOVE_ADDITIVE,
		MOVE_VELOCITY,
		MOVE_ABSOLUTE,
		MOVE_TORQUE,
		STOP_OFF,
		STOP_ON,
		HOME,
		POWER_OFF,
		POWER_ON,
		WAIT_FOR_ACTIVE,
		ERROR,
		ERROR_RESET,
		UPDATE,
		MOVE_OFF
		);
	HomingEnum :
		(
		PREPARE_HOME,
		HOMING,
		EXIT_HOME
		);
END_TYPE
```

### Program Logical/Source/Code/Logger/LoggerTask (IEC)

#### Types.typ
```iecst
TYPE
	LoggerHandlingType : 	STRUCT
		Input : LoggerHandlingInpType;
		Internal : LoggerHandlingInterType;
		Output : LoggerHandlingOutType;
	END_STRUCT;
END_TYPE

(**)

TYPE
	LoggerHandlingInpType : 	STRUCT
		Commands : LoggerHandlingInpCmdType;
		Parameters : LoggerHandlingInpParsType;
	END_STRUCT;
	LoggerHandlingInpCmdType : 	STRUCT
		GET_ID : BOOL;
		ERROR_RESET : BOOL;
		DELETE : BOOL;
		CREATE : BOOL;
		READ_DESC : BOOL;
		READ_ERROR_NUMBER : BOOL;
		READ : BOOL;
		GET_LATEST_RECORD : BOOL;
		GET_PREVIOUS : BOOL;
		ACK : BOOL;
		REL_START : BOOL;
	END_STRUCT;
	LoggerHandlingInpParsType : 	STRUCT
		NumberOfLogbook : USINT;
		NumberOfLog : INT;
		IDentLogToDelete : ArEventLogIdentType;
		NameOfNewLogbook : STRING[80];
		RecordID : UDINT;
		NameOfLogbook : STRING[80];
	END_STRUCT;
END_TYPE

(**)

TYPE
	LoggerHandlingInterType : 	STRUCT
		Fubs : LoggerHandlingInterFubsType;
		FuncAndParams : LoggerHandlingInterFuncAParsType;
	END_STRUCT;
	LoggerHandlingInterFubsType : 	STRUCT
		_ArEventLogCreate : ArEventLogCreate;
		_ArEventLogDelete : ArEventLogDelete;
		_ArEventLogGetIdent : ArEventLogGetIdent;
		_ArEventLogReadErrorNumber : ArEventLogReadErrorNumber;
		_ArEventLogReadDescription : ArEventLogReadDescription;
		_ArEventLogGetPreviousRecordID : ArEventLogGetPreviousRecordID;
		_ArEventLogGetLatestRecordID : ArEventLogGetLatestRecordID;
		_ArEventLogRead : ArEventLogRead;
		_ArEventLogReadObjectID : ArEventLogReadObjectID;
	END_STRUCT;
	LoggerHandlingInterFuncAParsType : 	STRUCT
		_ArEventLogIdentType : ArEventLogIdentType;
		_ArEventLogRecordIDType : ArEventLogRecordIDType;
		EventID : STRING[20];
		ConvTime : STRING[30];
		TimeLog : ArEventLogTimeStampType;
		TextBuffor : STRING[80];
		ErrorBuffor : STRING[30];
		ObjectID : STRING[36];
		i : UINT;
	END_STRUCT;
END_TYPE

(**)

TYPE
	LoggerHandlingOutType : 	STRUCT
		MainStep : MainStepEnum;
		ReadList : ReadErrorList;
		States : LoggerHandlingOutStatesType;
	END_STRUCT;
	LoggerHandlingOutStatesType : 	STRUCT
		LogList : STRING[450];
		LogDesc : STRING[1800];
		LogTime : STRING[1150];
		LogSeverity : STRING[150];
		EndStateCmd : STRING[80];
		FaultNumber : DINT;
		NumberOfFault : USINT;
	END_STRUCT;
END_TYPE

(**)

TYPE
	ReadErrorList :
		(
		START_REL,
		INIT_REL,
		GET_LATEST_REL,
		READ_REL,
		WAIT_FOR_EXE_REL,
		WAIT_FOR_DESC_REL,
		WAIT_FOR_ERROR_NUMBER_REL,
		CONVERSION_REL,
		NEXT_REL,
		ERROR_REL,
		END_REL
		);
	MainStepEnum :
		(
		WAIT_FOR_CMD_LH,
		CREATE_LOGBOOK_LH,
		GET_ID_LH,
		DELETE_LOGBOOK_LH,
		READ_LH,
		READ_ERROR_NUMBER_LH,
		READ_DESC_LH,
		ERROR_LH,
		ERROR_RESET_LH,
		GET_LATEST_RECORD_ID_LH,
		GET_PREVIOUS_RECORD_LH,
		ADD_TO_INTERNAL_LH,
		READ_OBJ_ID_LH
		);
END_TYPE
```

#### Variables.var
```iecst
VAR
	_LoggerHandling : LoggerHandlingType;
END_VAR
```

#### Main.st
```iecst
PROGRAM _INIT
	(* INIT INPUT PARAMETERS *)
	_LoggerHandling.Input.Parameters.NumberOfLog := 20;
	_LoggerHandling.Input.Parameters.NumberOfLogbook := 1;
	_LoggerHandling.Input.Parameters.NameOfLogbook := '$$arlogsys';
	_LoggerHandling.Input.Parameters.NameOfNewLogbook := 'UserLogbook';
	_LoggerHandling.Input.Parameters.RecordID := 10;
	_LoggerHandling.Internal.FuncAndParams.i := 0;
END_PROGRAM

PROGRAM _CYCLIC

	(*********************  MAIN STEP LIST  *********************)

	CASE _LoggerHandling.Output.MainStep OF
		WAIT_FOR_CMD_LH:
			IF _LoggerHandling.Input.Commands.GET_ID THEN
				_LoggerHandling.Input.Commands.GET_ID := FALSE;
				_LoggerHandling.Output.MainStep := GET_ID_LH;

			ELSIF _LoggerHandling.Input.Commands.CREATE THEN
				_LoggerHandling.Input.Commands.CREATE := FALSE;
				_LoggerHandling.Output.MainStep := CREATE_LOGBOOK_LH;

			ELSIF _LoggerHandling.Input.Commands.DELETE THEN
				_LoggerHandling.Input.Commands.DELETE := FALSE;
				_LoggerHandling.Output.MainStep := DELETE_LOGBOOK_LH;

			ELSIF _LoggerHandling.Input.Commands.READ THEN
				_LoggerHandling.Input.Commands.READ := FALSE;
				_LoggerHandling.Output.MainStep := READ_LH;

			ELSIF _LoggerHandling.Input.Commands.READ_DESC THEN
				_LoggerHandling.Input.Commands.READ_DESC := FALSE;
				_LoggerHandling.Output.MainStep := READ_DESC_LH;

			ELSIF _LoggerHandling.Input.Commands.READ_ERROR_NUMBER THEN
				_LoggerHandling.Input.Commands.READ_ERROR_NUMBER := FALSE;
				_LoggerHandling.Output.MainStep := READ_ERROR_NUMBER_LH;

			ELSIF _LoggerHandling.Input.Commands.GET_LATEST_RECORD THEN
				_LoggerHandling.Input.Commands.GET_LATEST_RECORD := FALSE;
				_LoggerHandling.Output.MainStep := GET_LATEST_RECORD_ID_LH;

			ELSIF _LoggerHandling.Input.Commands.GET_PREVIOUS THEN
				_LoggerHandling.Input.Commands.GET_PREVIOUS := FALSE;
				_LoggerHandling.Output.MainStep := GET_PREVIOUS_RECORD_LH;
			END_IF

		GET_ID_LH:
			_LoggerHandling.Internal.Fubs._ArEventLogGetIdent.Name 	  := _LoggerHandling.Input.Parameters.NameOfLogbook;
			_LoggerHandling.Internal.Fubs._ArEventLogGetIdent.Execute := TRUE;
			_LoggerHandling.Internal.Fubs._ArEventLogGetIdent();

			IF _LoggerHandling.Internal.Fubs._ArEventLogGetIdent.Done THEN
				_LoggerHandling.Internal.FuncAndParams._ArEventLogIdentType := _LoggerHandling.Internal.Fubs._ArEventLogGetIdent.Ident;
				_LoggerHandling.Internal.Fubs._ArEventLogGetIdent.Execute := FALSE;
				_LoggerHandling.Internal.Fubs._ArEventLogGetIdent();
				_LoggerHandling.Output.States.EndStateCmd := 'CMD_OK: GET ID';
				_LoggerHandling.Output.MainStep := WAIT_FOR_CMD_LH;

			ELSIF _LoggerHandling.Internal.Fubs._ArEventLogGetIdent.Error AND _LoggerHandling.Internal.Fubs._ArEventLogGetIdent.StatusID <> -1070586087 THEN

				_LoggerHandling.Output.States.EndStateCmd := 'CMD_ERROR: GET ID';
				_LoggerHandling.Output.States.FaultNumber := _LoggerHandling.Internal.Fubs._ArEventLogGetIdent.StatusID;
				_LoggerHandling.Internal.Fubs._ArEventLogGetIdent.Execute := FALSE;
				_LoggerHandling.Internal.Fubs._ArEventLogGetIdent();
				_LoggerHandling.Output.MainStep := ERROR_LH;

			ELSIF _LoggerHandling.Internal.Fubs._ArEventLogGetIdent.Error AND _LoggerHandling.Internal.Fubs._ArEventLogGetIdent.StatusID = -1070586087 THEN

				_LoggerHandling.Output.States.NumberOfFault := _LoggerHandling.Output.States.NumberOfFault +1;
				_LoggerHandling.Output.States.FaultNumber := _LoggerHandling.Internal.Fubs._ArEventLogGetIdent.StatusID;
				_LoggerHandling.Internal.Fubs._ArEventLogGetIdent.Execute := FALSE;
				_LoggerHandling.Internal.Fubs._ArEventLogGetIdent();
				_LoggerHandling.Output.States.EndStateCmd := 'CMD_ERROR: Logbook entry doesnt exist';
				_LoggerHandling.Output.MainStep := ERROR_LH;
			END_IF

		CREATE_LOGBOOK_LH:
			_LoggerHandling.Internal.Fubs._ArEventLogCreate.Execute := TRUE;
			_LoggerHandling.Internal.Fubs._ArEventLogCreate.Persistence := arEVENTLOG_PERSISTENCE_PERSIST;
			_LoggerHandling.Internal.Fubs._ArEventLogCreate.Size := 10000;
			_LoggerHandling.Internal.Fubs._ArEventLogCreate.Info := 0;
			_LoggerHandling.Internal.Fubs._ArEventLogCreate.Name := _LoggerHandling.Input.Parameters.NameOfNewLogbook;
			_LoggerHandling.Internal.Fubs._ArEventLogCreate();

			IF _LoggerHandling.Internal.Fubs._ArEventLogCreate.Done THEN
				_LoggerHandling.Internal.Fubs._ArEventLogCreate.Execute := FALSE;
				_LoggerHandling.Internal.Fubs._ArEventLogCreate();
				_LoggerHandling.Output.States.EndStateCmd := 'CMD_OK: CREATE LOGBOOK';
				_LoggerHandling.Output.MainStep := WAIT_FOR_CMD_LH;

			ELSIF _LoggerHandling.Internal.Fubs._ArEventLogCreate.Error THEN

				_LoggerHandling.Output.States.FaultNumber := _LoggerHandling.Internal.Fubs._ArEventLogCreate.StatusID;
				_LoggerHandling.Output.States.NumberOfFault := _LoggerHandling.Output.States.NumberOfFault+1;

				_LoggerHandling.Internal.Fubs._ArEventLogCreate.Execute := FALSE;
				_LoggerHandling.Internal.Fubs._ArEventLogCreate();
				_LoggerHandling.Output.States.EndStateCmd := 'CMD_ERROR: CREATE LOGBOOK';
				_LoggerHandling.Output.MainStep := ERROR_LH;
			END_IF

		DELETE_LOGBOOK_LH:
			_LoggerHandling.Internal.Fubs._ArEventLogDelete.Execute := TRUE;
			_LoggerHandling.Internal.Fubs._ArEventLogDelete.Ident := _LoggerHandling.Input.Parameters.IDentLogToDelete;
			_LoggerHandling.Internal.Fubs._ArEventLogDelete();

			IF   _LoggerHandling.Internal.Fubs._ArEventLogDelete.Done THEN
				_LoggerHandling.Internal.Fubs._ArEventLogDelete.Execute := FALSE;
				_LoggerHandling.Internal.Fubs._ArEventLogDelete();
				_LoggerHandling.Output.States.EndStateCmd := 'CMD_OK: DELETE LOGBOOK';
				_LoggerHandling.Output.MainStep := WAIT_FOR_CMD_LH;

			ELSIF _LoggerHandling.Internal.Fubs._ArEventLogDelete.Error THEN

				_LoggerHandling.Output.States.NumberOfFault := _LoggerHandling.Output.States.NumberOfFault +1;
				_LoggerHandling.Output.States.FaultNumber := _LoggerHandling.Internal.Fubs._ArEventLogDelete.StatusID;

				_LoggerHandling.Internal.Fubs._ArEventLogDelete.Execute := FALSE;
				_LoggerHandling.Internal.Fubs._ArEventLogDelete();
				_LoggerHandling.Output.States.EndStateCmd := 'CMD_ERROR: DELETE LOGBOOK';
				_LoggerHandling.Output.MainStep := ERROR_LH;
			END_IF;

		GET_LATEST_RECORD_ID_LH:
			_LoggerHandling.Internal.Fubs._ArEventLogGetLatestRecordID.Execute := TRUE;
			_LoggerHandling.Internal.Fubs._ArEventLogGetLatestRecordID.Ident := _LoggerHandling.Internal.FuncAndParams._ArEventLogIdentType;
			_LoggerHandling.Internal.Fubs._ArEventLogGetLatestRecordID();

			IF _LoggerHandling.Internal.Fubs._ArEventLogGetLatestRecordID.Done THEN
				_LoggerHandling.Internal.FuncAndParams._ArEventLogRecordIDType := _LoggerHandling.Internal.Fubs._ArEventLogGetLatestRecordID.RecordID;
				_LoggerHandling.Internal.Fubs._ArEventLogGetLatestRecordID.Execute := FALSE;
				_LoggerHandling.Internal.Fubs._ArEventLogGetLatestRecordID();
				_LoggerHandling.Output.States.EndStateCmd := 'CMD_OK: GET LATEST RECORD ID';
				_LoggerHandling.Output.MainStep := WAIT_FOR_CMD_LH;

			ELSIF _LoggerHandling.Internal.Fubs._ArEventLogGetLatestRecordID.Error THEN
				_LoggerHandling.Output.States.NumberOfFault := _LoggerHandling.Output.States.NumberOfFault +1;
				_LoggerHandling.Output.States.FaultNumber := _LoggerHandling.Internal.Fubs._ArEventLogGetLatestRecordID.StatusID;

				_LoggerHandling.Internal.Fubs._ArEventLogGetLatestRecordID.Execute := FALSE;
				_LoggerHandling.Internal.Fubs._ArEventLogGetLatestRecordID();
				_LoggerHandling.Output.States.EndStateCmd := 'CMD_ERROR: GET LATEST RECORD ID';
				_LoggerHandling.Output.MainStep := ERROR_LH;
			END_IF

		GET_PREVIOUS_RECORD_LH:
			_LoggerHandling.Internal.Fubs._ArEventLogGetPreviousRecordID.Execute := TRUE;
			_LoggerHandling.Internal.Fubs._ArEventLogGetPreviousRecordID.Ident := _LoggerHandling.Internal.FuncAndParams._ArEventLogIdentType;
			_LoggerHandling.Internal.Fubs._ArEventLogGetPreviousRecordID.RecordID := _LoggerHandling.Internal.FuncAndParams._ArEventLogRecordIDType;
			_LoggerHandling.Internal.Fubs._ArEventLogGetPreviousRecordID();

			IF _LoggerHandling.Internal.Fubs._ArEventLogGetPreviousRecordID.Done THEN
				_LoggerHandling.Internal.FuncAndParams._ArEventLogRecordIDType := _LoggerHandling.Internal.Fubs._ArEventLogGetPreviousRecordID.PrevRecordID;
				_LoggerHandling.Internal.Fubs._ArEventLogGetPreviousRecordID.Execute := FALSE;
				_LoggerHandling.Internal.Fubs._ArEventLogGetPreviousRecordID();
				_LoggerHandling.Output.States.EndStateCmd := 'CMD_OK: GET PREVIOUS RECORD';
				_LoggerHandling.Output.MainStep := WAIT_FOR_CMD_LH;

			ELSIF _LoggerHandling.Internal.Fubs._ArEventLogGetPreviousRecordID.Error AND _LoggerHandling.Internal.Fubs._ArEventLogGetPreviousRecordID.StatusID = -1070586096 THEN

				_LoggerHandling.Internal.Fubs._ArEventLogGetPreviousRecordID.Execute := FALSE;
				_LoggerHandling.Internal.Fubs._ArEventLogGetPreviousRecordID();
				_LoggerHandling.Output.States.EndStateCmd := 'CMD_DONE_ALL: GET PREVIOUS RECORD';
				_LoggerHandling.Output.MainStep := WAIT_FOR_CMD_LH;

			ELSIF _LoggerHandling.Internal.Fubs._ArEventLogGetPreviousRecordID.Error AND _LoggerHandling.Internal.Fubs._ArEventLogGetPreviousRecordID.StatusID <> -1070586096 THEN
				_LoggerHandling.Output.States.NumberOfFault := _LoggerHandling.Output.States.NumberOfFault +1;
				_LoggerHandling.Output.States.FaultNumber := _LoggerHandling.Internal.Fubs._ArEventLogGetPreviousRecordID.StatusID;

				_LoggerHandling.Internal.Fubs._ArEventLogGetPreviousRecordID.Execute := FALSE;
				_LoggerHandling.Internal.Fubs._ArEventLogGetPreviousRecordID();
				_LoggerHandling.Output.States.EndStateCmd := 'CMD_ERROR: GET PREVIOUS RECORD';
				_LoggerHandling.Output.MainStep := ERROR_LH;
			END_IF

		READ_LH:
			_LoggerHandling.Internal.Fubs._ArEventLogRead.Execute := TRUE;
			_LoggerHandling.Internal.Fubs._ArEventLogRead.Ident := _LoggerHandling.Internal.FuncAndParams._ArEventLogIdentType;
			_LoggerHandling.Internal.Fubs._ArEventLogRead.RecordID := _LoggerHandling.Internal.FuncAndParams._ArEventLogRecordIDType;
			_LoggerHandling.Internal.Fubs._ArEventLogRead();

			IF _LoggerHandling.Internal.Fubs._ArEventLogRead.Done THEN
				_LoggerHandling.Internal.FuncAndParams.EventID :=DINT_TO_STRING(_LoggerHandling.Internal.Fubs._ArEventLogRead.EventID);
				_LoggerHandling.Internal.FuncAndParams.TimeLog := _LoggerHandling.Internal.Fubs._ArEventLogRead.TimeStamp;
				_LoggerHandling.Internal.Fubs._ArEventLogRead.Execute := FALSE;
				_LoggerHandling.Internal.Fubs._ArEventLogRead();
				_LoggerHandling.Output.States.EndStateCmd := 'CMD_OK: READ';
				_LoggerHandling.Output.MainStep := WAIT_FOR_CMD_LH;

			ELSIF _LoggerHandling.Internal.Fubs._ArEventLogRead.Error THEN
				_LoggerHandling.Output.States.NumberOfFault := _LoggerHandling.Output.States.NumberOfFault +1;
				_LoggerHandling.Output.States.FaultNumber := _LoggerHandling.Internal.Fubs._ArEventLogRead.StatusID;

				_LoggerHandling.Internal.Fubs._ArEventLogRead.Execute := FALSE;
				_LoggerHandling.Internal.Fubs._ArEventLogRead();
				_LoggerHandling.Output.States.EndStateCmd := 'CMD_ERROR: READ';
				_LoggerHandling.Output.MainStep := ERROR_LH;
			END_IF

		READ_DESC_LH:
			_LoggerHandling.Internal.Fubs._ArEventLogReadDescription.Execute := TRUE;
			_LoggerHandling.Internal.Fubs._ArEventLogReadDescription.Ident := _LoggerHandling.Internal.FuncAndParams._ArEventLogIdentType;
			_LoggerHandling.Internal.Fubs._ArEventLogReadDescription.RecordID := _LoggerHandling.Internal.FuncAndParams._ArEventLogRecordIDType;
			_LoggerHandling.Internal.Fubs._ArEventLogReadDescription.LanguageCode := 'en';
			_LoggerHandling.Internal.Fubs._ArEventLogReadDescription.TextBuffer := ADR(_LoggerHandling.Internal.FuncAndParams.TextBuffor);
			_LoggerHandling.Internal.Fubs._ArEventLogReadDescription.TextBufferSize := 1000;
			_LoggerHandling.Internal.Fubs._ArEventLogReadDescription();

			IF _LoggerHandling.Internal.Fubs._ArEventLogReadDescription.Done THEN
				strcat(ADR(_LoggerHandling.Output.States.LogDesc),ADR(_LoggerHandling.Internal.FuncAndParams.TextBuffor));
				strcat(ADR(_LoggerHandling.Output.States.LogDesc),ADR(','));

				_LoggerHandling.Internal.Fubs._ArEventLogReadDescription.Execute := FALSE;
				_LoggerHandling.Internal.Fubs._ArEventLogReadDescription();
				_LoggerHandling.Output.States.EndStateCmd := 'CMD_OK: READ DESC';
				_LoggerHandling.Output.MainStep := WAIT_FOR_CMD_LH;

			ELSIF _LoggerHandling.Internal.Fubs._ArEventLogReadDescription.Error THEN
				_LoggerHandling.Output.States.NumberOfFault := _LoggerHandling.Output.States.NumberOfFault +1;
				_LoggerHandling.Output.States.FaultNumber := _LoggerHandling.Internal.Fubs._ArEventLogReadDescription.StatusID;

				_LoggerHandling.Internal.Fubs._ArEventLogReadDescription.Execute := FALSE;
				_LoggerHandling.Internal.Fubs._ArEventLogReadDescription();
				_LoggerHandling.Output.States.EndStateCmd := 'CMD_ERROR: READ DESC';
				_LoggerHandling.Output.MainStep := ERROR_LH;
			END_IF

		READ_ERROR_NUMBER_LH:
			_LoggerHandling.Internal.Fubs._ArEventLogReadErrorNumber.Execute := TRUE;
			_LoggerHandling.Internal.Fubs._ArEventLogReadErrorNumber.Ident := _LoggerHandling.Internal.FuncAndParams._ArEventLogIdentType;
			_LoggerHandling.Internal.Fubs._ArEventLogReadErrorNumber.RecordID := _LoggerHandling.Internal.FuncAndParams._ArEventLogRecordIDType;
			_LoggerHandling.Internal.Fubs._ArEventLogReadErrorNumber();

			IF _LoggerHandling.Internal.Fubs._ArEventLogReadErrorNumber.Error THEN

								_LoggerHandling.Output.States.NumberOfFault := _LoggerHandling.Output.States.NumberOfFault +1;
								_LoggerHandling.Output.States.FaultNumber := _LoggerHandling.Internal.Fubs._ArEventLogReadErrorNumber.StatusID;

								_LoggerHandling.Internal.Fubs._ArEventLogReadErrorNumber.Execute := FALSE;
								_LoggerHandling.Internal.Fubs._ArEventLogReadErrorNumber();
								_LoggerHandling.Output.States.EndStateCmd := 'CMD_ERROR: READ ERROR NUMBER';

								IF _LoggerHandling.Internal.FuncAndParams.i <> 0 THEN
									strcat(ADR(_LoggerHandling.Output.States.LogSeverity),ADR(',FA'));
								ELSE
									strcat(ADR(_LoggerHandling.Output.States.LogSeverity),ADR('FA'));
								END_IF

								_LoggerHandling.Output.MainStep := ERROR_LH;

			ELSIF _LoggerHandling.Internal.Fubs._ArEventLogReadErrorNumber.Done THEN

				_LoggerHandling.Internal.FuncAndParams.ErrorBuffor := UDINT_TO_STRING(_LoggerHandling.Internal.Fubs._ArEventLogReadErrorNumber.ErrorNumber);
				strcat(ADR(_LoggerHandling.Output.States.LogList),ADR(_LoggerHandling.Internal.FuncAndParams.ErrorBuffor));
				strcat(ADR(_LoggerHandling.Output.States.LogList),ADR(','));

				IF _LoggerHandling.Internal.FuncAndParams.i <> 0 THEN
					CASE _LoggerHandling.Internal.Fubs._ArEventLogReadErrorNumber.Severity OF
						arEVENTLOG_SEVERITY_SUCCESS:
							strcat(ADR(_LoggerHandling.Output.States.LogSeverity),ADR(',S'));
						arEVENTLOG_SEVERITY_INFO:
							strcat(ADR(_LoggerHandling.Output.States.LogSeverity),ADR(',I'));
						arEVENTLOG_SEVERITY_WARNING:
							strcat(ADR(_LoggerHandling.Output.States.LogSeverity),ADR(',W'));
						arEVENTLOG_SEVERITY_ERROR:
							strcat(ADR(_LoggerHandling.Output.States.LogSeverity),ADR(',E'));
						ELSE
							strcat(ADR(_LoggerHandling.Output.States.LogSeverity),ADR(',X'));
					END_CASE;
				ELSE
					CASE _LoggerHandling.Internal.Fubs._ArEventLogReadErrorNumber.Severity OF
						arEVENTLOG_SEVERITY_SUCCESS:
							strcat(ADR(_LoggerHandling.Output.States.LogSeverity),ADR('S'));
						arEVENTLOG_SEVERITY_INFO:
							strcat(ADR(_LoggerHandling.Output.States.LogSeverity),ADR('I'));
						arEVENTLOG_SEVERITY_WARNING:
							strcat(ADR(_LoggerHandling.Output.States.LogSeverity),ADR('W'));
						arEVENTLOG_SEVERITY_ERROR:
							strcat(ADR(_LoggerHandling.Output.States.LogSeverity),ADR('E'));
						ELSE
							strcat(ADR(_LoggerHandling.Output.States.LogSeverity),ADR('X'));
					END_CASE;
				END_IF

				_LoggerHandling.Internal.Fubs._ArEventLogReadErrorNumber.Execute := FALSE;
				_LoggerHandling.Internal.Fubs._ArEventLogReadErrorNumber();
				_LoggerHandling.Output.States.EndStateCmd := 'CMD_OK: READ ERROR NUMBER';
				_LoggerHandling.Output.MainStep := WAIT_FOR_CMD_LH;

			END_IF

		READ_OBJ_ID_LH:
			_LoggerHandling.Internal.Fubs._ArEventLogReadObjectID.Execute := TRUE;
			_LoggerHandling.Internal.Fubs._ArEventLogReadObjectID.Ident := _LoggerHandling.Internal.FuncAndParams._ArEventLogIdentType;
			_LoggerHandling.Internal.Fubs._ArEventLogReadObjectID.RecordID := _LoggerHandling.Internal.FuncAndParams._ArEventLogRecordIDType;
			_LoggerHandling.Internal.Fubs._ArEventLogReadObjectID();

			IF _LoggerHandling.Internal.Fubs._ArEventLogReadObjectID.Done THEN
				_LoggerHandling.Internal.FuncAndParams.ObjectID := _LoggerHandling.Internal.Fubs._ArEventLogReadObjectID.ObjectID;
				_LoggerHandling.Internal.Fubs._ArEventLogReadObjectID.Execute := FALSE;
				_LoggerHandling.Internal.Fubs._ArEventLogReadObjectID();
				_LoggerHandling.Output.States.EndStateCmd := 'CMD_OK: READ OBJ ID';
				_LoggerHandling.Output.MainStep := WAIT_FOR_CMD_LH;
			ELSIF _LoggerHandling.Internal.Fubs._ArEventLogReadObjectID.Error THEN
				_LoggerHandling.Output.States.NumberOfFault := _LoggerHandling.Output.States.NumberOfFault +1;
				_LoggerHandling.Output.States.FaultNumber := _LoggerHandling.Internal.Fubs._ArEventLogReadObjectID.StatusID;

				_LoggerHandling.Internal.Fubs._ArEventLogReadObjectID.Execute := FALSE;
				_LoggerHandling.Internal.Fubs._ArEventLogReadObjectID();
				_LoggerHandling.Output.States.EndStateCmd := 'CMD_ERROR: READ OBJ ID';
				_LoggerHandling.Output.MainStep := ERROR_LH;
			END_IF

		ADD_TO_INTERNAL_LH:
			_LoggerHandling.Internal.FuncAndParams._ArEventLogRecordIDType := _LoggerHandling.Input.Parameters.RecordID;
			_LoggerHandling.Output.MainStep := WAIT_FOR_CMD_LH;

		ERROR_LH:
			IF _LoggerHandling.Input.Commands.ERROR_RESET THEN
				_LoggerHandling.Input.Commands.ERROR_RESET := FALSE;
				_LoggerHandling.Output.MainStep := ERROR_RESET_LH;
			END_IF

		ERROR_RESET_LH:
			_LoggerHandling.Output.MainStep := WAIT_FOR_CMD_LH;
	END_CASE;

	(*********************  READ LIST CASE  *********************)

	CASE _LoggerHandling.Output.ReadList OF

		START_REL:
			_LoggerHandling.Output.States.EndStateCmd := 'NOT READ';
			IF _LoggerHandling.Input.Commands.REL_START THEN
				_LoggerHandling.Input.Commands.REL_START := FALSE;
				_LoggerHandling.Input.Commands.ACK := FALSE;
				_LoggerHandling.Internal.FuncAndParams.i := 0;
				_LoggerHandling.Output.States.LogDesc := '';
				_LoggerHandling.Output.States.LogList := '';
				_LoggerHandling.Output.States.LogSeverity := '';
				_LoggerHandling.Output.States.LogTime := '';
				_LoggerHandling.Output.States.FaultNumber := 0;
				_LoggerHandling.Output.States.NumberOfFault := 0;
				_LoggerHandling.Output.ReadList := INIT_REL;
			END_IF
		INIT_REL:
			_LoggerHandling.Input.Commands.GET_ID := TRUE;
			_LoggerHandling.Output.ReadList := GET_LATEST_REL;

		GET_LATEST_REL:
			IF _LoggerHandling.Output.MainStep = ERROR_LH THEN
				_LoggerHandling.Output.ReadList := ERROR_REL;

			ELSIF _LoggerHandling.Output.States.EndStateCmd = 'CMD_ERROR: Logbook entry doesnt exist' THEN
				_LoggerHandling.Output.ReadList := END_REL;

			ELSIF _LoggerHandling.Output.States.EndStateCmd = 'CMD_OK: GET ID' THEN
				_LoggerHandling.Input.Commands.GET_LATEST_RECORD := TRUE;
				_LoggerHandling.Output.ReadList := READ_REL;

			END_IF
		READ_REL:
			IF _LoggerHandling.Output.MainStep = ERROR_LH THEN
				_LoggerHandling.Output.ReadList := ERROR_REL;

			ELSIF _LoggerHandling.Output.States.EndStateCmd = 'CMD_OK: GET LATEST RECORD ID' OR _LoggerHandling.Output.States.EndStateCmd = 'CMD_OK: GET PREVIOUS RECORD'  THEN
				_LoggerHandling.Input.Commands.READ := TRUE;
				_LoggerHandling.Output.ReadList := WAIT_FOR_EXE_REL;

			ELSIF _LoggerHandling.Output.States.EndStateCmd = 'CMD_DONE_ALL: GET PREVIOUS RECORD' THEN
				_LoggerHandling.Output.ReadList := END_REL;
			END_IF

		WAIT_FOR_EXE_REL:
			IF _LoggerHandling.Output.MainStep = ERROR_LH THEN
				_LoggerHandling.Output.ReadList := ERROR_REL;

			ELSIF _LoggerHandling.Output.States.EndStateCmd = 'CMD_OK: READ' THEN

				IF _LoggerHandling.Internal.FuncAndParams.EventID <> '0' THEN

					strcat(ADR(_LoggerHandling.Output.States.LogList),ADR(_LoggerHandling.Internal.FuncAndParams.EventID));
					strcat(ADR(_LoggerHandling.Output.States.LogList),ADR(','));
					_LoggerHandling.Input.Commands.READ_DESC := TRUE;
					_LoggerHandling.Output.ReadList := WAIT_FOR_DESC_REL;

				ELSE

					_LoggerHandling.Input.Commands.READ_ERROR_NUMBER := TRUE;
					_LoggerHandling.Output.ReadList := WAIT_FOR_ERROR_NUMBER_REL;
				END_IF
			END_IF

		WAIT_FOR_ERROR_NUMBER_REL:
			IF  _LoggerHandling.Output.MainStep = ERROR_LH  THEN
				_LoggerHandling.Output.ReadList := ERROR_REL;

			ELSIF _LoggerHandling.Output.States.EndStateCmd = 'CMD_OK: READ ERROR NUMBER' THEN
				_LoggerHandling.Input.Commands.READ_DESC := TRUE;
				_LoggerHandling.Output.ReadList := WAIT_FOR_DESC_REL;

			END_IF

		WAIT_FOR_DESC_REL:
			IF  _LoggerHandling.Output.MainStep = ERROR_LH  THEN
				_LoggerHandling.Output.ReadList := ERROR_REL;

			ELSIF _LoggerHandling.Output.States.EndStateCmd = 'CMD_OK: READ DESC' THEN
				_LoggerHandling.Output.ReadList := CONVERSION_REL;
			END_IF

		CONVERSION_REL:
			_LoggerHandling.Internal.FuncAndParams.ConvTime := DT_TO_STRING(DATE_TO_DT(UDINT_TO_DATE(_LoggerHandling.Internal.FuncAndParams.TimeLog.sec + 3600 +(_LoggerHandling.Internal.FuncAndParams.TimeLog.nsec/1000000000))));

			strcat(ADR(_LoggerHandling.Output.States.LogTime),ADR(_LoggerHandling.Internal.FuncAndParams.ConvTime));
			strcat(ADR(_LoggerHandling.Output.States.LogTime),ADR(','));

			_LoggerHandling.Output.ReadList := NEXT_REL;

		NEXT_REL:

			_LoggerHandling.Internal.FuncAndParams.i := _LoggerHandling.Internal.FuncAndParams.i + 1;

			IF _LoggerHandling.Internal.FuncAndParams.i >= _LoggerHandling.Input.Parameters.NumberOfLog THEN
				_LoggerHandling.Output.States.EndStateCmd := 'CMD_OK: READING_ALL_LOG_DONE';
				_LoggerHandling.Output.ReadList := END_REL;
			ELSE
				_LoggerHandling.Input.Commands.GET_PREVIOUS := TRUE;
				_LoggerHandling.Output.ReadList := READ_REL;
			END_IF

		END_REL:
			IF _LoggerHandling.Input.Commands.ACK THEN
				_LoggerHandling.Input.Commands.ACK := FALSE;
				_LoggerHandling.Output.ReadList := START_REL;
			END_IF

		ERROR_REL:
			IF _LoggerHandling.Input.Commands.ACK THEN
				_LoggerHandling.Input.Commands.ERROR_RESET := TRUE;
				_LoggerHandling.Output.ReadList := START_REL;
			END_IF
	END_CASE;

END_PROGRAM

PROGRAM _EXIT

END_PROGRAM
```

### Program Logical/Source/Code/Memory/MemTask (IEC)

#### Types.typ
```iecst
TYPE
	MemTaskType : 	STRUCT
		Input : MemTaskInputType;
		Internal : MemTaskInterType;
		Output : MemTaskOutputType;
	END_STRUCT;
END_TYPE

(**)

TYPE
	MemTaskInputType : 	STRUCT
		Cmd : MemTaskInputCmdType;
		Params : MemTaskInputParmsType;
	END_STRUCT;
END_TYPE

(**)

TYPE
	MemTaskInputCmdType : 	STRUCT
		Start : BOOL;
		RepeatAll : BOOL;
		ReapetOnce : BOOL;
		Ack : BOOL;
	END_STRUCT;
	MemTaskInputParmsType : 	STRUCT
		MemType : USINT;
	END_STRUCT;
END_TYPE

(**)

TYPE
	MemTaskInterType : 	STRUCT
		memXInfo : MEMxInfo;
		memBuffor : STRING[20];
		iter : USINT;
	END_STRUCT;
END_TYPE

(**)

TYPE
	MemTaskOutputType : 	STRUCT
		States : MemTaskOutputStatesType;
		MemStateMachine : MemoryTaskEnum;
	END_STRUCT;
	MemTaskOutputStatesType : 	STRUCT
		Status : STRING[20];
		brUSRROM : STRING[50];
		brUSRRAM : STRING[50];
		brSYSROM : STRING[50];
		brDRAM : STRING[50];
	END_STRUCT;
END_TYPE

(**)

TYPE
	MemoryTaskEnum :
		(
		WAIT_FOR_CMD_MT,
		START_MT,
		READ_ONCE_MT,
		READ_MT,
		WRITE_IN_OUTPUT_MT,
		DONE_MT
		);
END_TYPE
```

#### Variables.var
```iecst
VAR
	_MemTask : MemTaskType;
END_VAR
```

#### Main.st
```iecst
PROGRAM _INIT
	(*
0 ... brDRAM (TMP_Ram)
1 ... brUSRRAM (USR_Ram)
2 ... brSYSROM (SYS_Prom)
3 ... brUSRROM (USR_Prom)
 *)

END_PROGRAM

PROGRAM _CYCLIC
	CASE _MemTask.Output.MemStateMachine OF
		WAIT_FOR_CMD_MT:
			IF _MemTask.Input.Cmd.Start THEN
				_MemTask.Input.Cmd.Start := FALSE;
				_MemTask.Output.MemStateMachine := START_MT;
			ELSIF _MemTask.Input.Cmd.RepeatAll THEN
				_MemTask.Input.Cmd.RepeatAll := FALSE;
				_MemTask.Output.MemStateMachine := START_MT;
			ELSIF _MemTask.Input.Cmd.ReapetOnce THEN
				_MemTask.Input.Cmd.ReapetOnce := FALSE;
				_MemTask.Internal.memXInfo.mem_typ := _MemTask.Input.Params.MemType;
				_MemTask.Output.MemStateMachine := READ_MT;
			END_IF
			_MemTask.Output.States.Status := 'WAIT_FOR_CMD';

		START_MT:
			_MemTask.Internal.iter := 0;
			_MemTask.Internal.memXInfo.enable := TRUE;
			_MemTask.Internal.memXInfo.mem_typ := _MemTask.Internal.iter;
			_MemTask.Output.MemStateMachine := READ_MT;

			_MemTask.Output.States.brDRAM 	:= '';
			_MemTask.Output.States.brUSRRAM := '';
			_MemTask.Output.States.brUSRROM := '';
			_MemTask.Output.States.brSYSROM := '';
			_MemTask.Output.States.Status 	:= 'START';

		READ_MT:
			_MemTask.Internal.memXInfo();

			IF _MemTask.Internal.memXInfo.status = ERR_OK THEN

					CASE _MemTask.Internal.iter OF
					0:
						_MemTask.Internal.memBuffor := UDINT_TO_STRING(_MemTask.Internal.memXInfo.MemSize);
						strcat(ADR(_MemTask.Output.States.brDRAM),ADR(_MemTask.Internal.memBuffor));
						strcat(ADR(_MemTask.Output.States.brDRAM),ADR('|'));
						_MemTask.Internal.memBuffor := UDINT_TO_STRING(_MemTask.Internal.memXInfo.FreeMemSize);
						strcat(ADR(_MemTask.Output.States.brDRAM),ADR(_MemTask.Internal.memBuffor));
						strcat(ADR(_MemTask.Output.States.brDRAM),ADR('|'));
						_MemTask.Internal.memBuffor := UDINT_TO_STRING(_MemTask.Internal.memXInfo.BiggestFreeBlockSize);
						strcat(ADR(_MemTask.Output.States.brDRAM),ADR(_MemTask.Internal.memBuffor));
					1:
						_MemTask.Internal.memBuffor := UDINT_TO_STRING(_MemTask.Internal.memXInfo.MemSize);
						strcat(ADR(_MemTask.Output.States.brUSRRAM),ADR(_MemTask.Internal.memBuffor));
						strcat(ADR(_MemTask.Output.States.brUSRRAM),ADR('|'));
						_MemTask.Internal.memBuffor := UDINT_TO_STRING(_MemTask.Internal.memXInfo.FreeMemSize);
						strcat(ADR(_MemTask.Output.States.brUSRRAM),ADR(_MemTask.Internal.memBuffor));
						strcat(ADR(_MemTask.Output.States.brUSRRAM),ADR('|'));
						_MemTask.Internal.memBuffor := UDINT_TO_STRING(_MemTask.Internal.memXInfo.BiggestFreeBlockSize);
						strcat(ADR(_MemTask.Output.States.brUSRRAM),ADR(_MemTask.Internal.memBuffor));
					2:
						_MemTask.Internal.memBuffor := UDINT_TO_STRING(_MemTask.Internal.memXInfo.MemSize);
						strcat(ADR(_MemTask.Output.States.brSYSROM),ADR(_MemTask.Internal.memBuffor));
						strcat(ADR(_MemTask.Output.States.brSYSROM),ADR('|'));
						_MemTask.Internal.memBuffor := UDINT_TO_STRING(_MemTask.Internal.memXInfo.FreeMemSize);
						strcat(ADR(_MemTask.Output.States.brSYSROM),ADR(_MemTask.Internal.memBuffor));
						strcat(ADR(_MemTask.Output.States.brSYSROM),ADR('|'));
						_MemTask.Internal.memBuffor := UDINT_TO_STRING(_MemTask.Internal.memXInfo.BiggestFreeBlockSize);
						strcat(ADR(_MemTask.Output.States.brSYSROM),ADR(_MemTask.Internal.memBuffor));
					3:
						_MemTask.Internal.memBuffor := UDINT_TO_STRING(_MemTask.Internal.memXInfo.MemSize);
						strcat(ADR(_MemTask.Output.States.brUSRROM),ADR(_MemTask.Internal.memBuffor));
						strcat(ADR(_MemTask.Output.States.brUSRROM),ADR('|'));
						_MemTask.Internal.memBuffor := UDINT_TO_STRING(_MemTask.Internal.memXInfo.FreeMemSize);
						strcat(ADR(_MemTask.Output.States.brUSRROM),ADR(_MemTask.Internal.memBuffor));
						strcat(ADR(_MemTask.Output.States.brUSRROM),ADR('|'));
						_MemTask.Internal.memBuffor := UDINT_TO_STRING(_MemTask.Internal.memXInfo.BiggestFreeBlockSize);
						strcat(ADR(_MemTask.Output.States.brUSRROM),ADR(_MemTask.Internal.memBuffor));
				END_CASE;
				_MemTask.Output.MemStateMachine := WRITE_IN_OUTPUT_MT;
			END_IF

		READ_ONCE_MT:
			_MemTask.Internal.memXInfo.mem_typ := _MemTask.Input.Params.MemType;
			_MemTask.Internal.memXInfo();

			IF _MemTask.Internal.memXInfo.status = ERR_OK THEN

				_MemTask.Output.MemStateMachine := WRITE_IN_OUTPUT_MT;
			END_IF

		WRITE_IN_OUTPUT_MT:
			_MemTask.Internal.iter := _MemTask.Internal.iter +1;

			IF _MemTask.Internal.iter > 3 THEN
				_MemTask.Internal.iter := 0;
				_MemTask.Output.MemStateMachine := DONE_MT;
			ELSE
				_MemTask.Internal.memXInfo.mem_typ := _MemTask.Internal.iter;
				_MemTask.Output.MemStateMachine := READ_MT;

			END_IF

		DONE_MT:
			_MemTask.Output.States.Status := 'MemTest: DONE';
			IF _MemTask.Input.Cmd.Ack THEN
				_MemTask.Input.Cmd.Ack := FALSE;
				_MemTask.Output.MemStateMachine := WAIT_FOR_CMD_MT;
			END_IF

	END_CASE;

END_PROGRAM

PROGRAM _EXIT
	(* Insert code here *)

END_PROGRAM
```

### Program Logical/Source/Code/Controller/ControllerTask (IEC)

#### Types.typ
```iecst
TYPE
	ControllerType : 	STRUCT
		Input : ControllerInputType;
		Internal : ControllerInternalType;
		Output : ControllerOutputType;
	END_STRUCT;
END_TYPE

(**)

TYPE
	ControllerInputType : 	STRUCT
		Cmd : ControllerInpCmdType;
		Params : ControllerInpParamsType;
	END_STRUCT;
	ControllerInternalType : 	STRUCT
		Fubs : ControllerFubsType;
	END_STRUCT;
	ControllerOutputType : 	STRUCT
		Time : DATE_AND_TIME;
		ProjectInfo : ControllerOutputProjInfoType;
	END_STRUCT;
	ControllerOutputProjInfoType : 	STRUCT
		ConfigurationVersion : STRING[64];
		ConfigurationID : STRING[255];
		Done : BOOL;
		ErrorID : DINT;
	END_STRUCT;
END_TYPE

(**)

TYPE
	ControllerInpCmdType : 	STRUCT
		DoReset : BOOL;
		GetInfoAboutProject : BOOL;
		GetTime : BOOL;
	END_STRUCT;
	ControllerInpParamsType : 	STRUCT
		ResetType : USINT;
	END_STRUCT;
END_TYPE

(**)

TYPE
	ControllerFubsType : 	STRUCT
		ProjectGetInfo : ArProjectGetInfo;
		GetTime : DTGetTime;
	END_STRUCT;
END_TYPE
```

#### Variables.var
```iecst
VAR
	_Controller : ControllerType;
END_VAR
```

#### Main.st
```iecst
PROGRAM _INIT
	_Controller.Input.Params.ResetType := 0;

END_PROGRAM

PROGRAM _CYCLIC
	(************************** Get time **************************)
	_Controller.Internal.Fubs.GetTime.enable := _Controller.Input.Cmd.GetTime;

	IF _Controller.Internal.Fubs.GetTime.status = ERR_OK AND _Controller.Input.Cmd.GetTime THEN
		_Controller.Output.Time := _Controller.Internal.Fubs.GetTime.DT1;
	END_IF
	_Controller.Internal.Fubs.GetTime();
	(**************************          **************************)

	(************************** Reset systemu **************************)
	SYSreset(_Controller.Input.Cmd.DoReset,_Controller.Input.Params.ResetType);
	(**************************               **************************)

	(************************** Project info **************************)
	IF _Controller.Input.Cmd.GetInfoAboutProject THEN
		_Controller.Internal.Fubs.ProjectGetInfo.Execute := TRUE;

		IF _Controller.Internal.Fubs.ProjectGetInfo.Done THEN
			_Controller.Input.Cmd.GetInfoAboutProject := FALSE;
			_Controller.Output.ProjectInfo.ConfigurationID := _Controller.Internal.Fubs.ProjectGetInfo.ConfigurationID;
			_Controller.Output.ProjectInfo.ConfigurationVersion := _Controller.Internal.Fubs.ProjectGetInfo.ConfigurationVersion;
			_Controller.Output.ProjectInfo.Done := TRUE;

			_Controller.Internal.Fubs.ProjectGetInfo.Execute := FALSE;
			_Controller.Internal.Fubs.ProjectGetInfo();

		ELSIF _Controller.Internal.Fubs.ProjectGetInfo.Error THEN
			_Controller.Internal.Fubs.ProjectGetInfo.Execute := FALSE;
			_Controller.Output.ProjectInfo.ErrorID := _Controller.Internal.Fubs.ProjectGetInfo.StatusID;
			_Controller.Output.ProjectInfo.Done := TRUE;
			_Controller.Internal.Fubs.ProjectGetInfo();
		END_IF
		_Controller.Internal.Fubs.ProjectGetInfo();
	END_IF
	(**************************              **************************)

	(** TODO: BRSystem,Zmiana adresu IP sterownika **)

END_PROGRAM

PROGRAM _EXIT
	(* Insert code here *)

END_PROGRAM
```

### Program Logical/Source/Code/Chart/ChartTask (IEC)

#### Types.typ
```iecst
TYPE
	TraceType : 	STRUCT
		Input : TraceInpType;
		Internal : TraceIntType;
		Output : TraceOutType;
	END_STRUCT;
END_TYPE

(**)

TYPE
	TraceInpType : 	STRUCT
		Cmd : TraceInpCmdType;
		Params : TraceInpParmsType;
	END_STRUCT;
	TraceInpCmdType : 	STRUCT
		Start : BOOL;
		ResetError : BOOL;
	END_STRUCT;
	TraceInpParmsType : 	STRUCT
		NumberOfParams : BOOL;
		NameOfParams : STRING[80];
	END_STRUCT;
END_TYPE

(**)

TYPE
	TraceIntType : 	STRUCT
		Fubs : TraceIntFubsType;
		Func : TraceIntFuncType;
		Params : TraceIntParamsType;
	END_STRUCT;
	TraceIntFubsType : 	STRUCT
		Fileread : FileRead;
		Fileopen : FileOpen;
		ParTrace : MC_BR_ParTrace;
	END_STRUCT;
	TraceIntFuncType : 	STRUCT
		PARTRACECONFIG : MC_PARTRACECONFIG_REF;
	END_STRUCT;
	TraceIntParamsType : 	STRUCT
		FileLenght : REAL;
		Offset : UDINT;
		VlvTrans : STRING[15];
		Iteration : INT;
		ParamsIn : STRING[1000];
	END_STRUCT;
END_TYPE

(**)

TYPE
	TraceOutType : 	STRUCT
		StateMachine : TraceSM;
		Status : TraceOutStatusType;
	END_STRUCT;
	TraceOutStatusType : 	STRUCT
		ParamsOut : STRING[1000];
		ErrorStatus : USINT;
	END_STRUCT;
	TraceSM :
		(
		WAIT_FOR_CMD_T,
		START_T,
		READ_T,
		ERROR_RESET_T,
		ERROR_T,
		OPEN_T,
		WAIT_FOR_READ_T,
		CONNECT_TXT_T
		);
END_TYPE
```

#### Variables.var
```iecst
VAR
	_Trace : TraceType;
END_VAR
```

#### Main.st
```iecst
PROGRAM _INIT

//	_Trace.Internal.Fubs.ReadNetTraceStatus.Enable := TRUE;
//	_Trace.Internal.Fubs.ReadNetTraceStatus.Configuration := ;
//
//	_Trace.Internal.Fubs.ReadParTraceStatus.Enable := TRUE;
//	_Trace.Internal.Fubs.ReadParTraceStatus.Configuration := ;

	// ACP10PAR_SCTRL_SPEED_ACT ;
	//	ACP10PAR_ENCOD1_S_ACT
				//	ACP10PAR_PCTRL_S_ACT
				//	ACP10PAR_TORQUE_ACT
				//	ACP10PAR_

	_Trace.Internal.Params.Offset := 0;
END_PROGRAM

PROGRAM _CYCLIC

	CASE _Trace.Output.StateMachine OF
		WAIT_FOR_CMD_T:

			IF _Trace.Input.Cmd.Start THEN
				_Trace.Input.Cmd.Start := FALSE;
				_Trace.Output.StateMachine := START_T;
			END_IF

		START_T:
			IF NOT _Trace.Internal.Fubs.ParTrace.Busy AND NOT _Trace.Internal.Fubs.ParTrace.Done THEN
				_Trace.Internal.Func.PARTRACECONFIG.DatObj.Device := 'AppSave';
				_Trace.Internal.Func.PARTRACECONFIG.DatObj.Format := mcFILE_TXT;
				_Trace.Internal.Func.PARTRACECONFIG.DatObj.Name   := 'chartAutoApp';
				_Trace.Internal.Func.PARTRACECONFIG.DatObj.Type   := mcFILE;

				_Trace.Internal.Func.PARTRACECONFIG.ParTrace.SamplingTime := 0.1;
				_Trace.Internal.Func.PARTRACECONFIG.ParTrace.TracingTime  := 15;
				_Trace.Internal.Func.PARTRACECONFIG.ParTrace.Type := mcMULTI_AXIS_TRACE;
				_Trace.Internal.Func.PARTRACECONFIG.ParTrace.Delay := 0;
				_Trace.Internal.Func.PARTRACECONFIG.ParTrace.NetTriggerDelay := 0;
				_Trace.Internal.Func.PARTRACECONFIG.ParTrace.Trigger.Threshold := 90;

				_Trace.Internal.Func.PARTRACECONFIG.ParTrace.Parameter[0].Axis  := ADR(gAxis01);
				_Trace.Internal.Func.PARTRACECONFIG.ParTrace.Parameter[0].ParID := ACP10PAR_PCTRL_V_ACT;

			END_IF

			_Trace.Internal.Fubs.ParTrace.Execute := TRUE;
			_Trace.Internal.Fubs.ParTrace.Command := mcSTART+mcSAVE;
			_Trace.Internal.Fubs.ParTrace.Configuration := _Trace.Internal.Func.PARTRACECONFIG;
			_Trace.Internal.Fubs.ParTrace();

			IF _Trace.Internal.Fubs.ParTrace.Done THEN
				_Trace.Internal.Fubs.ParTrace.Execute := FALSE;
				_Trace.Internal.Fubs.ParTrace();
				_Trace.Output.StateMachine := OPEN_T;

			ELSIF _Trace.Internal.Fubs.ParTrace.Error THEN
				_Trace.Output.StateMachine := ERROR_T;

			END_IF

		OPEN_T:
			_Trace.Internal.Fubs.Fileopen.enable  := TRUE;
			_Trace.Internal.Fubs.Fileopen.mode 	  := fiREAD_ONLY;
			_Trace.Internal.Fubs.Fileopen.pDevice := ADR('AppSave');
			_Trace.Internal.Fubs.Fileopen.pFile   := ADR('\chartAutoApp.txt');
			_Trace.Internal.Fubs.Fileopen();

			IF _Trace.Internal.Fubs.Fileopen.status = ERR_OK THEN
				_Trace.Internal.Fubs.Fileread.ident := _Trace.Internal.Fubs.Fileopen.ident;
				_Trace.Internal.Params.FileLenght 	:= _Trace.Internal.Fubs.Fileopen.filelen;

				_Trace.Internal.Fubs.Fileopen.enable := FALSE;
				_Trace.Internal.Fubs.Fileopen();
				_Trace.Output.StateMachine := READ_T;
			ELSIF _Trace.Internal.Fubs.Fileopen.status <> ERR_OK AND NOT _Trace.Internal.Fubs.Fileopen.status = ERR_FUB_BUSY THEN

				_Trace.Internal.Fubs.Fileopen.enable := FALSE;
				_Trace.Output.StateMachine := ERROR_T;

			ELSIF _Trace.Internal.Fubs.Fileopen.status = ERR_FUB_BUSY THEN

			END_IF
		READ_T:
			_Trace.Internal.Fubs.Fileread.enable := TRUE;
			_Trace.Internal.Fubs.Fileread.pDest  := ADR(_Trace.Internal.Params.ParamsIn);
			_Trace.Internal.Fubs.Fileread.len 	 := 1000;
			_Trace.Internal.Fubs.Fileread.offset := _Trace.Internal.Params.Offset;
			_Trace.Internal.Fubs.Fileread();
			// $r$n
			IF _Trace.Internal.Fubs.Fileread.status = ERR_OK THEN
				_Trace.Internal.Fubs.Fileread.enable := FALSE;
				_Trace.Internal.Fubs.Fileread();

				_Trace.Output.StateMachine := CONNECT_TXT_T;
			END_IF

		CONNECT_TXT_T:
		//	FOR _Trace.Internal.Params.Iteration = 0

		WAIT_FOR_READ_T:

		ERROR_T:

		ERROR_RESET_T:

	END_CASE;

END_PROGRAM

PROGRAM _EXIT
	(* Insert code here *)

END_PROGRAM
```

### Data object Logical/acp10etxen (Ett)

- acp10etxen.ett (not shown)

### Package Logical/gAxis01obj - gAxis01obj

### gAxis01a.apt
```
AcoposParameterTable:
  Root Parameters
```

### gAxis01i.ax
```
InitParameter (Version=3.18.2, NcSwId=Acp10)
  ACP10AXIS_typ:
    dig_in:
      level:
        reference = ncACTIV_HI
        pos_hw_end = ncACTIV_HI
        neg_hw_end = ncACTIV_HI
        trigger1 = ncACTIV_HI
        trigger2 = ncACTIV_HI
    encoder_if:
      parameter:
        count_dir = ncSTANDARD
        scaling:
          load:
            units = 1000
            rev_motor = 1
    limit:
      parameter:
        v_pos = 10000
        v_neg = 10000
        a1_pos = 50000
        a2_pos = 50000
        a1_neg = 50000
        a2_neg = 50000
        t_jolt = 0
        t_in_pos = 0
        pos_sw_end = 2000000000
        neg_sw_end = -2000000000
        ds_warning = 500
        ds_stop = 1000
        a_stop = 1.0e30
        dv_stop = 0
        dv_stop_mode = ncOFF
    controller:
      mode = ncPOSITION
      position:
        kv = 50
        tn = 0
        t_predict = 0.0004
        t_total = 0.0004
        p_max = 1.0e30
        i_max = 0
      speed:
        kv = 2.0
        tn = 0
        t_filter = 0.0
        isq_filter1:
          type = ncOFF
          a0 = 0.0
          a1 = 0.0
          b0 = 0.0
          b1 = 0.0
          b2 = 0.0
          c0_par_id = 0
          c1_par_id = 0
        isq_filter2:
          type = ncOFF
          a0 = 0.0
          a1 = 0.0
          b0 = 0.0
          b1 = 0.0
          b2 = 0.0
          c0_par_id = 0
          c1_par_id = 0
        isq_filter3:
          type = ncOFF
          a0 = 0.0
          a1 = 0.0
          b0 = 0.0
          b1 = 0.0
          b2 = 0.0
          c0_par_id = 0
          c1_par_id = 0
      uf:
        type = ncLINEAR
        auto_config = ncMOTOR_PAR
        u0 = 0
        un = 0
        fn = 50.0
        k_f_slip = 0
      ff:
        torque_load = 0.0
        torque_pos = 0.0
        torque_neg = 0.0
        kv_torque = 0.0
        inertia = 0.0
        t_filter_a = 0.0
    move:
      stop:
        parameter[0]:
          decel_ramp = ncA_LIMIT
          controller = ncON
        parameter[1]:
          decel_ramp = ncA_LIMIT
          controller = ncON
        parameter[2]:
          decel_ramp = ncA_LIMIT
          controller = ncON
        parameter[3]:
          decel_ramp = ncA_LIMIT
          controller = ncON
        quickstop:
          decel_ramp = ncA_LIMIT
        drive_error:
          decel_ramp = ncA_LIMIT
      homing:
        parameter:
          s = 0
          v_switch = 5000
          v_trigger = 500
          a = 50000
          mode = ncDIRECT
          edge_sw = ncPOSITIVE
          start_dir = ncPOSITIVE
          trigg_dir = ncPOSITIVE
          ref_pulse = ncOFF
          fix_dir = ncOFF
          tr_s_block = 0
          torque_lim = 0
          ds_block = 0
          ds_stop = 0
      basis:
        parameter:
          v_pos = 5000
          v_neg = 5000
          a1_pos = 50000
          a2_pos = 50000
          a1_neg = 50000
          a2_neg = 50000
    message:
      text:
        parameter:
          format = ncBREAK
          columns = 80
          data_modul = acp10etxen
```
